LIN {X 0,Y 554.453,Z 809.786,A -85,B 0,C 180,E1 23627.307,E2 23627.307} C_VEL
LIN {X 0,Y 557.118,Z 789.157,A -85,B 0,C 180,E1 23626.499,E2 23626.499} C_VEL
LIN {X 0,Y 559.409,Z 768.857,A -85,B 0,C 180,E1 23625.833,E2 23625.833} C_VEL
LIN {X 0,Y 561.829,Z 743.404,A -85,B 0,C 180,E1 23625.168,E2 23625.168} C_VEL
LIN {X 0,Y 563.453,Z 718.234,A -85,B 0,C 180,E1 23624.694,E2 23624.694} C_VEL
LIN {X 0,Y 571.021,Z 495.759,A -85,B 0,C 180,E1 23621.491,E2 23621.491} C_VEL
LIN {X 0,Y 575.269,Z 370.947,A -85,B 0,C 180,E1 23619.667,E2 23619.667} C_VEL
LIN {X 0,Y 560.09,Z 346.765,A -85,B 0,C 180,E1 23617.356,E2 23617.356} C_VEL
LIN {X 0,Y 547.087,Z 327.659,A -85,B 0,C 180,E1 23615.214,E2 23615.214} C_VEL
LIN {X 0,Y 534.986,Z 310.945,A -85,B 0,C 180,E1 23613.044,E2 23613.044} C_VEL
LIN {X 0,Y 528.375,Z 302.282,A -85,B 0,C 180,E1 23611.773,E2 23611.773} C_VEL
LIN {X 0,Y 524.681,Z 297.482,A -85,B 0,C 180,E1 23611.031,E2 23611.031} C_VEL
LIN {X 0,Y 520.373,Z 291.905,A -85,B 0,C 180,E1 23610.132,E2 23610.132} C_VEL
LIN {X 0,Y 514.951,Z 285.155,A -85,B 0,C 180,E1 23608.914,E2 23608.914} C_VEL
LIN {X 0,Y 513.768,Z 282.099,A -85,B 0,C 180,E1 23608.162,E2 23608.162} C_VEL
LIN {X 0,Y 513.798,Z 281.966,A -85,B 0,C 180,E1 23604.857,E2 23604.857} C_VEL
LIN {X 0,Y 513.742,Z 281.98,A -85,B 0,C 180,E1 23601.583,E2 23601.583} C_VEL
LIN {X 0,Y 513.762,Z 281.984,A -85,B 0,C 180,E1 23598.143,E2 23598.143} C_VEL
LIN {X 0,Y 513.802,Z 281.979,A -85,B 0,C 180,E1 23594.719,E2 23594.719} C_VEL
LIN {X 0,Y 513.743,Z 281.974,A -85,B 0,C 180,E1 23591.337,E2 23591.337} C_VEL
LIN {X 0,Y 513.747,Z 281.962,A -85,B 0,C 180,E1 23587.83,E2 23587.83} C_VEL
LIN {X 0,Y 513.79,Z 281.955,A -85,B 0,C 180,E1 23584.577,E2 23584.577} C_VEL
LIN {X 0,Y 513.742,Z 281.977,A -85,B 0,C 180,E1 23581.227,E2 23581.227} C_VEL
LIN {X 0,Y 513.756,Z 281.987,A -85,B 0,C 180,E1 23577.769,E2 23577.769} C_VEL
LIN {X 0,Y 513.801,Z 281.966,A -85,B 0,C 180,E1 23574.304,E2 23574.304} C_VEL
LIN {X 0,Y 513.739,Z 281.958,A -85,B 0,C 180,E1 23571.042,E2 23571.042} C_VEL
LIN {X 0,Y 513.749,Z 281.959,A -85,B 0,C 180,E1 23567.524,E2 23567.524} C_VEL
LIN {X 0,Y 513.799,Z 281.966,A -85,B 0,C 180,E1 23564.19,E2 23564.19} C_VEL
LIN {X 0,Y 513.746,Z 281.987,A -85,B 0,C 180,E1 23560.797,E2 23560.797} C_VEL
LIN {X 0,Y 513.747,Z 281.987,A -85,B 0,C 180,E1 23557.213,E2 23557.213} C_VEL
LIN {X 0,Y 513.787,Z 281.879,A -85,B 0,C 180,E1 23553.907,E2 23553.907} C_VEL
LIN {X 0,Y 513.743,Z 281.964,A -85,B 0,C 180,E1 23550.629,E2 23550.629} C_VEL
LIN {X 0,Y 513.776,Z 282.125,A -85,B 0,C 180,E1 23548.389,E2 23548.389} C_VEL
LIN {X 0,Y 514.13,Z 283.467,A -85,B 0,C 180,E1 23548.085,E2 23548.085} C_VEL
LIN {X 0,Y 516.016,Z 286.518,A -85,B 0,C 180,E1 23547.636,E2 23547.636} C_VEL
LIN {X 0,Y 518.738,Z 288.732,A -85,B 0,C 180,E1 23547.073,E2 23547.073} C_VEL
LIN {X 0,Y 521.096,Z 292.417,A -85,B 0,C 180,E1 23546.552,E2 23546.552} C_VEL
LIN {X 0,Y 523.689,Z 294.869,A -85,B 0,C 180,E1 23546.033,E2 23546.033} C_VEL
LIN {X 0,Y 526.696,Z 298.998,A -85,B 0,C 180,E1 23545.415,E2 23545.415} C_VEL
LIN {X 0,Y 528.665,Z 301.077,A -85,B 0,C 180,E1 23545.035,E2 23545.035} C_VEL
LIN {X 0,Y 532.356,Z 305.607,A -85,B 0,C 180,E1 23544.324,E2 23544.324} C_VEL
LIN {X 0,Y 537,Z 311.379,A -85,B 0,C 180,E1 23543.461,E2 23543.461} C_VEL
LIN {X 0,Y 547.46,Z 325.856,A -85,B 0,C 180,E1 23541.594,E2 23541.594} C_VEL
LIN {X 0,Y 559.237,Z 342.837,A -85,B 0,C 180,E1 23539.649,E2 23539.649} C_VEL
LIN {X 0,Y 572.432,Z 363.406,A -85,B 0,C 180,E1 23537.625,E2 23537.625} C_VEL
LIN {X 0,Y 575.353,Z 368.355,A -85,B 0,C 180,E1 23537.193,E2 23537.193} C_VEL
LIN {X 0,Y 568.04,Z 579.703,A -85,B 0,C 180,E1 23534.136,E2 23534.136} C_VEL
LIN {X 0,Y 563.485,Z 712.252,A -85,B 0,C 180,E1 23532.221,E2 23532.221} C_VEL
LIN {X 0,Y 561.614,Z 739.268,A -85,B 0,C 180,E1 23531.688,E2 23531.688} C_VEL
LIN {X 0,Y 559.393,Z 762.648,A -85,B 0,C 180,E1 23531.056,E2 23531.056} C_VEL
LIN {X 0,Y 557.101,Z 783.032,A -85,B 0,C 180,E1 23530.373,E2 23530.373} C_VEL
LIN {X 0,Y 555.447,Z 790.439,A -85,B 0,C 180,E1 23530.171,E2 23530.171} C_VEL
LIN {X 0,Y 548.34,Z 809.024,A -85,B 0,C 180,E1 23529.808,E2 23529.808} C_VEL
LIN {X 0,Y 546.528,Z 815.961,A -85,B 0,C 180,E1 23529.545,E2 23529.545} C_VEL
LIN {X 0,Y 542.785,Z 839.215,A -85,B 0,C 180,E1 23528.327,E2 23528.327} C_VEL
LIN {X 0,Y 538.67,Z 861.769,A -85,B 0,C 180,E1 23526.911,E2 23526.911} C_VEL
LIN {X 0,Y 535.119,Z 880.065,A -85,B 0,C 180,E1 23525.595,E2 23525.595} C_VEL
LIN {X 0,Y 530.917,Z 900.978,A -85,B 0,C 180,E1 23523.88,E2 23523.88} C_VEL
LIN {X 0,Y 526.661,Z 920.781,A -85,B 0,C 180,E1 23521.985,E2 23521.985} C_VEL
LIN {X 0,Y 523.184,Z 936.83,A -85,B 0,C 180,E1 23520.248,E2 23520.248} C_VEL
LIN {X 0,Y 519.3,Z 954.991,A -85,B 0,C 180,E1 23518.022,E2 23518.022} C_VEL
LIN {X 0,Y 515.864,Z 971.093,A -85,B 0,C 180,E1 23515.733,E2 23515.733} C_VEL
LIN {X 0,Y 513.206,Z 984.016,A -85,B 0,C 180,E1 23513.663,E2 23513.663} C_VEL
LIN {X 0,Y 510.445,Z 998.558,A -85,B 0,C 180,E1 23511.006,E2 23511.006} C_VEL
LIN {X 0,Y 508.335,Z 1010.476,A -85,B 0,C 180,E1 23508.462,E2 23508.462} C_VEL
LIN {X 0,Y 506.857,Z 1020.106,A -85,B 0,C 180,E1 23506.112,E2 23506.112} C_VEL
LIN {X 0,Y 505.518,Z 1030.455,A -85,B 0,C 180,E1 23503.148,E2 23503.148} C_VEL
LIN {X 0,Y 504.78,Z 1037.728,A -85,B 0,C 180,E1 23500.615,E2 23500.615} C_VEL
LIN {X 0,Y 504.322,Z 1043.483,A -85,B 0,C 180,E1 23498.207,E2 23498.207} C_VEL
LIN {X 0,Y 504.05,Z 1048.716,A -85,B 0,C 180,E1 23495.464,E2 23495.464} C_VEL
LIN {X 0,Y 503.926,Z 1052.486,A -85,B 0,C 180,E1 23492.616,E2 23492.616} C_VEL
LIN {X 0,Y 503.916,Z 1054.489,A -85,B 0,C 180,E1 23490.227,E2 23490.227} C_VEL
LIN {X 0,Y 503.906,Z 1055.407,A -85,B 0,C 180,E1 23487.953,E2 23487.953} C_VEL
LIN {X 0,Y 503.904,Z 1055.329,A -85,B 0,C 180,E1 23485.562,E2 23485.562} C_VEL
LIN {X 0,Y 503.914,Z 1053.882,A -85,B 0,C 180,E1 23482.704,E2 23482.704} C_VEL
LIN {X 0,Y 503.979,Z 1050.859,A -85,B 0,C 180,E1 23479.945,E2 23479.945} C_VEL
LIN {X 0,Y 504.123,Z 1047.055,A -85,B 0,C 180,E1 23477.514,E2 23477.514} C_VEL
LIN {X 0,Y 504.455,Z 1041.841,A -85,B 0,C 180,E1 23474.95,E2 23474.95} C_VEL
LIN {X 0,Y 505.157,Z 1033.874,A -85,B 0,C 180,E1 23471.895,E2 23471.895} C_VEL
LIN {X 0,Y 506.062,Z 1025.946,A -85,B 0,C 180,E1 23469.409,E2 23469.409} C_VEL
LIN {X 0,Y 507.375,Z 1016.657,A -85,B 0,C 180,E1 23466.91,E2 23466.91} C_VEL
LIN {X 0,Y 509.449,Z 1003.972,A -85,B 0,C 180,E1 23464.016,E2 23464.016} C_VEL
LIN {X 0,Y 511.536,Z 992.584,A -85,B 0,C 180,E1 23461.769,E2 23461.769} C_VEL
LIN {X 0,Y 514.287,Z 978.894,A -85,B 0,C 180,E1 23459.377,E2 23459.377} C_VEL
LIN {X 0,Y 517.779,Z 962.343,A -85,B 0,C 180,E1 23456.873,E2 23456.873} C_VEL
LIN {X 0,Y 520.999,Z 947.641,A -85,B 0,C 180,E1 23454.915,E2 23454.915} C_VEL
LIN {X 0,Y 524.8,Z 930.682,A -85,B 0,C 180,E1 23452.906,E2 23452.906} C_VEL
LIN {X 0,Y 529.269,Z 910.241,A -85,B 0,C 180,E1 23450.807,E2 23450.807} C_VEL
LIN {X 0,Y 533.009,Z 892.867,A -85,B 0,C 180,E1 23449.245,E2 23449.245} C_VEL
LIN {X 0,Y 537.423,Z 871.919,A -85,B 0,C 180,E1 23447.59,E2 23447.59} C_VEL
LIN {X 0,Y 541.641,Z 850.035,A -85,B 0,C 180,E1 23446.117,E2 23446.117} C_VEL
LIN {X 0,Y 545.084,Z 830.856,A -85,B 0,C 180,E1 23444.997,E2 23444.997} C_VEL
LIN {X 0,Y 548.736,Z 808.878,A -85,B 0,C 180,E1 23443.891,E2 23443.891} C_VEL
LIN {X 0,Y 552.207,Z 784.715,A -85,B 0,C 180,E1 23442.885,E2 23442.885} C_VEL
LIN {X 0,Y 554.847,Z 763.158,A -85,B 0,C 180,E1 23442.15,E2 23442.15} C_VEL
LIN {X 0,Y 557.173,Z 740.46,A -85,B 0,C 180,E1 23441.525,E2 23441.525} C_VEL
LIN {X 0,Y 559.277,Z 712.892,A -85,B 0,C 180,E1 23440.968,E2 23440.968} C_VEL
LIN {X 0,Y 563.361,Z 607.457,A -85,B 0,C 180,E1 23439.413,E2 23439.413} C_VEL
LIN {X 0,Y 571.302,Z 402.325,A -85,B 0,C 180,E1 23436.395,E2 23436.395} C_VEL
LIN {X 0,Y 572.427,Z 372.307,A -85,B 0,C 180,E1 23435.938,E2 23435.938} C_VEL
LIN {X 0,Y 562.587,Z 356.836,A -85,B 0,C 180,E1 23434.292,E2 23434.292} C_VEL
LIN {X 0,Y 552.342,Z 341.781,A -85,B 0,C 180,E1 23432.463,E2 23432.463} C_VEL
LIN {X 0,Y 541.602,Z 326.838,A -85,B 0,C 180,E1 23430.388,E2 23430.388} C_VEL
LIN {X 0,Y 534.491,Z 317.842,A -85,B 0,C 180,E1 23428.92,E2 23428.92} C_VEL
LIN {X 0,Y 530.838,Z 313.286,A -85,B 0,C 180,E1 23428.124,E2 23428.124} C_VEL
LIN {X 0,Y 527.164,Z 308.769,A -85,B 0,C 180,E1 23427.293,E2 23427.293} C_VEL
LIN {X 0,Y 522.625,Z 303.55,A -85,B 0,C 180,E1 23426.229,E2 23426.229} C_VEL
LIN {X 0,Y 521.397,Z 301.779,A -85,B 0,C 180,E1 23425.92,E2 23425.92} C_VEL
LIN {X 0,Y 518.037,Z 298.4,A -85,B 0,C 180,E1 23425.097,E2 23425.097} C_VEL
LIN {X 0,Y 516.427,Z 295.827,A -85,B 0,C 180,E1 23424.661,E2 23424.661} C_VEL
LIN {X 0,Y 513.235,Z 293.149,A -85,B 0,C 180,E1 23423.845,E2 23423.845} C_VEL
LIN {X 0,Y 511.085,Z 289.592,A -85,B 0,C 180,E1 23423.217,E2 23423.217} C_VEL
LIN {X 0,Y 507.836,Z 287.317,A -85,B 0,C 180,E1 23422.334,E2 23422.334} C_VEL
LIN {X 0,Y 506.002,Z 283.836,A -85,B 0,C 180,E1 23421.686,E2 23421.686} C_VEL
LIN {X 0,Y 505.81,Z 282.987,A -85,B 0,C 180,E1 23421.208,E2 23421.208} C_VEL
LIN {X 0,Y 505.854,Z 282.932,A -85,B 0,C 180,E1 23417.841,E2 23417.841} C_VEL
LIN {X 0,Y 505.802,Z 282.897,A -85,B 0,C 180,E1 23414.54,E2 23414.54} C_VEL
LIN {X 0,Y 505.804,Z 282.954,A -85,B 0,C 180,E1 23411.055,E2 23411.055} C_VEL
LIN {X 0,Y 505.863,Z 282.882,A -85,B 0,C 180,E1 23407.724,E2 23407.724} C_VEL
LIN {X 0,Y 505.812,Z 282.949,A -85,B 0,C 180,E1 23404.308,E2 23404.308} C_VEL
LIN {X 0,Y 505.793,Z 282.891,A -85,B 0,C 180,E1 23400.793,E2 23400.793} C_VEL
LIN {X 0,Y 505.852,Z 282.939,A -85,B 0,C 180,E1 23397.508,E2 23397.508} C_VEL
LIN {X 0,Y 505.802,Z 282.898,A -85,B 0,C 180,E1 23394.214,E2 23394.214} C_VEL
LIN {X 0,Y 505.799,Z 282.933,A -85,B 0,C 180,E1 23390.671,E2 23390.671} C_VEL
LIN {X 0,Y 505.849,Z 282.89,A -85,B 0,C 180,E1 23387.326,E2 23387.326} C_VEL
LIN {X 0,Y 505.807,Z 282.926,A -85,B 0,C 180,E1 23384.051,E2 23384.051} C_VEL
LIN {X 0,Y 505.8,Z 282.897,A -85,B 0,C 180,E1 23380.553,E2 23380.553} C_VEL
LIN {X 0,Y 505.867,Z 282.942,A -85,B 0,C 180,E1 23377.206,E2 23377.206} C_VEL
LIN {X 0,Y 505.888,Z 283.351,A -85,B 0,C 180,E1 23375.667,E2 23375.667} C_VEL
LIN {X 0,Y 506.575,Z 285.399,A -85,B 0,C 180,E1 23375.17,E2 23375.17} C_VEL
LIN {X 0,Y 508.745,Z 288.207,A -85,B 0,C 180,E1 23374.505,E2 23374.505} C_VEL
LIN {X 0,Y 510.733,Z 289.915,A -85,B 0,C 180,E1 23373.958,E2 23373.958} C_VEL
LIN {X 0,Y 514.994,Z 294.989,A -85,B 0,C 180,E1 23372.791,E2 23372.791} C_VEL
LIN {X 0,Y 520.334,Z 301.55,A -85,B 0,C 180,E1 23371.413,E2 23371.413} C_VEL
LIN {X 0,Y 524.051,Z 305.988,A -85,B 0,C 180,E1 23370.51,E2 23370.51} C_VEL
LIN {X 0,Y 533.967,Z 318.851,A -85,B 0,C 180,E1 23368.251,E2 23368.251} C_VEL
LIN {X 0,Y 541.359,Z 328.901,A -85,B 0,C 180,E1 23366.7,E2 23366.7} C_VEL
LIN {X 0,Y 550.777,Z 341.951,A -85,B 0,C 180,E1 23364.866,E2 23364.866} C_VEL
LIN {X 0,Y 563.419,Z 360.814,A -85,B 0,C 180,E1 23362.599,E2 23362.599} C_VEL
LIN {X 0,Y 572.579,Z 375.694,A -85,B 0,C 180,E1 23361.069,E2 23361.069} C_VEL
LIN {X 0,Y 563.489,Z 607.493,A -85,B 0,C 180,E1 23357.666,E2 23357.666} C_VEL
LIN {X 0,Y 559.152,Z 720.201,A -85,B 0,C 180,E1 23356.004,E2 23356.004} C_VEL
LIN {X 0,Y 557.029,Z 747.91,A -85,B 0,C 180,E1 23355.449,E2 23355.449} C_VEL
LIN {X 0,Y 554.683,Z 770.486,A -85,B 0,C 180,E1 23354.834,E2 23354.834} C_VEL
LIN {X 0,Y 552.215,Z 790.549,A -85,B 0,C 180,E1 23354.16,E2 23354.16} C_VEL
LIN {X 0,Y 548.962,Z 813.722,A -85,B 0,C 180,E1 23353.224,E2 23353.224} C_VEL
LIN {X 0,Y 545.173,Z 836.653,A -85,B 0,C 180,E1 23352.094,E2 23352.094} C_VEL
LIN {X 0,Y 541.804,Z 855.478,A -85,B 0,C 180,E1 23351.017,E2 23351.017} C_VEL
LIN {X 0,Y 538.226,Z 874.224,A -85,B 0,C 180,E1 23349.791,E2 23349.791} C_VEL
LIN {X 0,Y 533.578,Z 897.113,A -85,B 0,C 180,E1 23348.062,E2 23348.062} C_VEL
LIN {X 0,Y 529.676,Z 915.321,A -85,B 0,C 180,E1 23346.469,E2 23346.469} C_VEL
LIN {X 0,Y 525.936,Z 932.493,A -85,B 0,C 180,E1 23344.774,E2 23344.774} C_VEL
LIN {X 0,Y 521.701,Z 951.969,A -85,B 0,C 180,E1 23342.586,E2 23342.586} C_VEL
LIN {X 0,Y 518.183,Z 968.123,A -85,B 0,C 180,E1 23340.496,E2 23340.496} C_VEL
LIN {X 0,Y 515.146,Z 982.591,A -85,B 0,C 180,E1 23338.394,E2 23338.394} C_VEL
LIN {X 0,Y 511.931,Z 998.836,A -85,B 0,C 180,E1 23335.696,E2 23335.696} C_VEL
LIN {X 0,Y 509.659,Z 1011.141,A -85,B 0,C 180,E1 23333.341,E2 23333.341} C_VEL
LIN {X 0,Y 507.902,Z 1021.942,A -85,B 0,C 180,E1 23330.996,E2 23330.996} C_VEL
LIN {X 0,Y 506.189,Z 1033.931,A -85,B 0,C 180,E1 23327.948,E2 23327.948} C_VEL
LIN {X 0,Y 505.253,Z 1042.032,A -85,B 0,C 180,E1 23325.495,E2 23325.495} C_VEL
LIN {X 0,Y 504.615,Z 1048.867,A -85,B 0,C 180,E1 23323.055,E2 23323.055} C_VEL
LIN {X 0,Y 504.158,Z 1055.624,A -85,B 0,C 180,E1 23320.051,E2 23320.051} C_VEL
LIN {X 0,Y 504,Z 1059.867,A -85,B 0,C 180,E1 23317.524,E2 23317.524} C_VEL
LIN {X 0,Y 503.923,Z 1062.669,A -85,B 0,C 180,E1 23315.237,E2 23315.237} C_VEL
LIN {X 0,Y 503.915,Z 1064.536,A -85,B 0,C 180,E1 23312.843,E2 23312.843} C_VEL
LIN {X 0,Y 503.913,Z 1065.403,A -85,B 0,C 180,E1 23310,E2 23310} C_VEL
LIN {X 0,Y 503.914,Z 1064.536,A -85,B 0,C 180,E1 23307.157,E2 23307.157} C_VEL
LIN {X 0,Y 503.923,Z 1062.669,A -85,B 0,C 180,E1 23304.763,E2 23304.763} C_VEL
LIN {X 0,Y 504.005,Z 1059.707,A -85,B 0,C 180,E1 23302.362,E2 23302.362} C_VEL
LIN {X 0,Y 504.219,Z 1054.753,A -85,B 0,C 180,E1 23299.488,E2 23299.488} C_VEL
LIN {X 0,Y 504.663,Z 1048.26,A -85,B 0,C 180,E1 23296.713,E2 23296.713} C_VEL
LIN {X 0,Y 505.289,Z 1041.681,A -85,B 0,C 180,E1 23294.388,E2 23294.388} C_VEL
LIN {X 0,Y 506.319,Z 1033.012,A -85,B 0,C 180,E1 23291.786,E2 23291.786} C_VEL
LIN {X 0,Y 507.978,Z 1021.444,A -85,B 0,C 180,E1 23288.887,E2 23288.887} C_VEL
LIN {X 0,Y 509.666,Z 1011.134,A -85,B 0,C 180,E1 23286.653,E2 23286.653} C_VEL
LIN {X 0,Y 511.933,Z 998.852,A -85,B 0,C 180,E1 23284.304,E2 23284.304} C_VEL
LIN {X 0,Y 515.136,Z 982.53,A -85,B 0,C 180,E1 23281.605,E2 23281.605} C_VEL
LIN {X 0,Y 517.974,Z 968.796,A -85,B 0,C 180,E1 23279.618,E2 23279.618} C_VEL
LIN {X 0,Y 521.233,Z 953.482,A -85,B 0,C 180,E1 23277.642,E2 23277.642} C_VEL
LIN {X 0,Y 525.45,Z 933.627,A -85,B 0,C 180,E1 23275.402,E2 23275.402} C_VEL
LIN {X 0,Y 529.03,Z 916.65,A -85,B 0,C 180,E1 23273.731,E2 23273.731} C_VEL
LIN {X 0,Y 532.787,Z 898.489,A -85,B 0,C 180,E1 23272.144,E2 23272.144} C_VEL
LIN {X 0,Y 537.401,Z 875.144,A -85,B 0,C 180,E1 23270.38,E2 23270.38} C_VEL
LIN {X 0,Y 540.935,Z 855.93,A -85,B 0,C 180,E1 23269.13,E2 23269.13} C_VEL
LIN {X 0,Y 544.258,Z 836.615,A -85,B 0,C 180,E1 23268.032,E2 23268.032} C_VEL
LIN {X 0,Y 548.122,Z 811.924,A -85,B 0,C 180,E1 23266.837,E2 23266.837} C_VEL
LIN {X 0,Y 551.03,Z 790.28,A -85,B 0,C 180,E1 23265.974,E2 23265.974} C_VEL
LIN {X 0,Y 553.399,Z 770.117,A -85,B 0,C 180,E1 23265.303,E2 23265.303} C_VEL
LIN {X 0,Y 555.717,Z 746.778,A -85,B 0,C 180,E1 23264.675,E2 23264.675} C_VEL
LIN {X 0,Y 557.645,Z 719.813,A -85,B 0,C 180,E1 23264.145,E2 23264.145} C_VEL
LIN {X 0,Y 562.993,Z 569.232,A -85,B 0,C 180,E1 23261.957,E2 23261.957} C_VEL
LIN {X 0,Y 569.951,Z 374.77,A -85,B 0,C 180,E1 23259.119,E2 23259.119} C_VEL
LIN {X 0,Y 555.897,Z 352.262,A -85,B 0,C 180,E1 23256.925,E2 23256.925} C_VEL
LIN {X 0,Y 543.365,Z 333.687,A -85,B 0,C 180,E1 23254.814,E2 23254.814} C_VEL
LIN {X 0,Y 531.41,Z 317,A -85,B 0,C 180,E1 23252.621,E2 23252.621} C_VEL
LIN {X 0,Y 524.88,Z 308.402,A -85,B 0,C 180,E1 23251.337,E2 23251.337} C_VEL
LIN {X 0,Y 521.584,Z 304.102,A -85,B 0,C 180,E1 23250.659,E2 23250.659} C_VEL
LIN {X 0,Y 517.442,Z 298.685,A -85,B 0,C 180,E1 23249.777,E2 23249.777} C_VEL
LIN {X 0,Y 509.213,Z 288.567,A -85,B 0,C 180,E1 23247.925,E2 23247.925} C_VEL
LIN {X 0,Y 506.669,Z 285.635,A -85,B 0,C 180,E1 23247.312,E2 23247.312} C_VEL
LIN {X 0,Y 505.899,Z 283.213,A -85,B 0,C 180,E1 23246.784,E2 23246.784} C_VEL
LIN {X 0,Y 505.807,Z 282.953,A -85,B 0,C 180,E1 23243.474,E2 23243.474} C_VEL
LIN {X 0,Y 505.805,Z 282.952,A -85,B 0,C 180,E1 23239.878,E2 23239.878} C_VEL
LIN {X 0,Y 505.857,Z 282.943,A -85,B 0,C 180,E1 23236.533,E2 23236.533} C_VEL
LIN {X 0,Y 505.808,Z 282.954,A -85,B 0,C 180,E1 23233.257,E2 23233.257} C_VEL
LIN {X 0,Y 505.807,Z 282.967,A -85,B 0,C 180,E1 23229.788,E2 23229.788} C_VEL
LIN {X 0,Y 505.871,Z 282.967,A -85,B 0,C 180,E1 23226.469,E2 23226.469} C_VEL
LIN {X 0,Y 505.811,Z 282.958,A -85,B 0,C 180,E1 23223.06,E2 23223.06} C_VEL
LIN {X 0,Y 505.801,Z 282.948,A -85,B 0,C 180,E1 23219.547,E2 23219.547} C_VEL
LIN {X 0,Y 505.854,Z 282.945,A -85,B 0,C 180,E1 23216.26,E2 23216.26} C_VEL
LIN {X 0,Y 505.81,Z 282.971,A -85,B 0,C 180,E1 23212.909,E2 23212.909} C_VEL
LIN {X 0,Y 505.807,Z 282.976,A -85,B 0,C 180,E1 23209.406,E2 23209.406} C_VEL
LIN {X 0,Y 505.864,Z 282.949,A -85,B 0,C 180,E1 23206.046,E2 23206.046} C_VEL
LIN {X 0,Y 505.814,Z 282.947,A -85,B 0,C 180,E1 23202.633,E2 23202.633} C_VEL
LIN {X 0,Y 505.802,Z 282.948,A -85,B 0,C 180,E1 23199.155,E2 23199.155} C_VEL
LIN {X 0,Y 505.852,Z 282.915,A -85,B 0,C 180,E1 23195.847,E2 23195.847} C_VEL
LIN {X 0,Y 505.807,Z 282.879,A -85,B 0,C 180,E1 23192.446,E2 23192.446} C_VEL
LIN {X 0,Y 505.885,Z 283.108,A -85,B 0,C 180,E1 23189.964,E2 23189.964} C_VEL
LIN {X 0,Y 506.188,Z 284.461,A -85,B 0,C 180,E1 23189.644,E2 23189.644} C_VEL
LIN {X 0,Y 507.959,Z 287.469,A -85,B 0,C 180,E1 23189.183,E2 23189.183} C_VEL
LIN {X 0,Y 510.968,Z 289.763,A -85,B 0,C 180,E1 23188.517,E2 23188.517} C_VEL
LIN {X 0,Y 513.385,Z 293.549,A -85,B 0,C 180,E1 23187.945,E2 23187.945} C_VEL
LIN {X 0,Y 515.995,Z 295.955,A -85,B 0,C 180,E1 23187.388,E2 23187.388} C_VEL
LIN {X 0,Y 518.916,Z 299.969,A -85,B 0,C 180,E1 23186.747,E2 23186.747} C_VEL
LIN {X 0,Y 520.905,Z 301.993,A -85,B 0,C 180,E1 23186.34,E2 23186.34} C_VEL
LIN {X 0,Y 524.449,Z 306.505,A -85,B 0,C 180,E1 23185.61,E2 23185.61} C_VEL
LIN {X 0,Y 526.85,Z 309.592,A -85,B 0,C 180,E1 23185.129,E2 23185.129} C_VEL
LIN {X 0,Y 530.776,Z 314.451,A -85,B 0,C 180,E1 23184.368,E2 23184.368} C_VEL
LIN {X 0,Y 536.926,Z 322.269,A -85,B 0,C 180,E1 23183.222,E2 23183.222} C_VEL
LIN {X 0,Y 547.877,Z 337.772,A -85,B 0,C 180,E1 23181.279,E2 23181.279} C_VEL
LIN {X 0,Y 558.734,Z 354.056,A -85,B 0,C 180,E1 23179.487,E2 23179.487} C_VEL
LIN {X 0,Y 569.982,Z 371.818,A -85,B 0,C 180,E1 23177.754,E2 23177.754} C_VEL
LIN {X 0,Y 562.566,Z 578.071,A -85,B 0,C 180,E1 23174.749,E2 23174.749} C_VEL
LIN {X 0,Y 557.767,Z 712.284,A -85,B 0,C 180,E1 23172.796,E2 23172.796} C_VEL
LIN {X 0,Y 555.852,Z 739.196,A -85,B 0,C 180,E1 23172.263,E2 23172.263} C_VEL
LIN {X 0,Y 553.559,Z 762.585,A -85,B 0,C 180,E1 23171.628,E2 23171.628} C_VEL
LIN {X 0,Y 551.1,Z 783.671,A -85,B 0,C 180,E1 23170.918,E2 23170.918} C_VEL
LIN {X 0,Y 547.756,Z 808.18,A -85,B 0,C 180,E1 23169.914,E2 23169.914} C_VEL
LIN {X 0,Y 546.528,Z 815.961,A -85,B 0,C 180,E1 23169.545,E2 23169.545} C_VEL
LIN {X 0,Y 544.695,Z 823.17,A -85,B 0,C 180,E1 23169.267,E2 23169.267} C_VEL
LIN {X 0,Y 537.052,Z 841.058,A -85,B 0,C 180,E1 23168.715,E2 23168.715} C_VEL
LIN {X 0,Y 535.041,Z 847.674,A -85,B 0,C 180,E1 23168.378,E2 23168.378} C_VEL
LIN {X 0,Y 531.464,Z 866.376,A -85,B 0,C 180,E1 23167.151,E2 23167.151} C_VEL
LIN {X 0,Y 526.686,Z 889.643,A -85,B 0,C 180,E1 23165.382,E2 23165.382} C_VEL
LIN {X 0,Y 522.685,Z 908.053,A -85,B 0,C 180,E1 23163.756,E2 23163.756} C_VEL
LIN {X 0,Y 518.678,Z 926.111,A -85,B 0,C 180,E1 23161.949,E2 23161.949} C_VEL
LIN {X 0,Y 514.32,Z 945.439,A -85,B 0,C 180,E1 23159.719,E2 23159.719} C_VEL
LIN {X 0,Y 510.958,Z 960.33,A -85,B 0,C 180,E1 23157.758,E2 23157.758} C_VEL
LIN {X 0,Y 507.691,Z 975.222,A -85,B 0,C 180,E1 23155.551,E2 23155.551} C_VEL
LIN {X 0,Y 504.387,Z 990.91,A -85,B 0,C 180,E1 23152.864,E2 23152.864} C_VEL
LIN {X 0,Y 502.139,Z 1002.299,A -85,B 0,C 180,E1 23150.626,E2 23150.626} C_VEL
LIN {X 0,Y 500.194,Z 1013.298,A -85,B 0,C 180,E1 23148.17,E2 23148.17} C_VEL
LIN {X 0,Y 498.438,Z 1024.538,A -85,B 0,C 180,E1 23145.222,E2 23145.222} C_VEL
LIN {X 0,Y 497.418,Z 1032.418,A -85,B 0,C 180,E1 23142.775,E2 23142.775} C_VEL
LIN {X 0,Y 496.721,Z 1039.128,A -85,B 0,C 180,E1 23140.32,E2 23140.32} C_VEL
LIN {X 0,Y 496.214,Z 1045.826,A -85,B 0,C 180,E1 23137.293,E2 23137.293} C_VEL
LIN {X 0,Y 496.013,Z 1050.189,A -85,B 0,C 180,E1 23134.625,E2 23134.625} C_VEL
LIN {X 0,Y 495.927,Z 1052.949,A -85,B 0,C 180,E1 23132.311,E2 23132.311} C_VEL
LIN {X 0,Y 495.929,Z 1054.797,A -85,B 0,C 180,E1 23129.884,E2 23129.884} C_VEL
LIN {X 0,Y 495.901,Z 1055.675,A -85,B 0,C 180,E1 23126.995,E2 23126.995} C_VEL
LIN {X 0,Y 495.917,Z 1054.841,A -85,B 0,C 180,E1 23124.098,E2 23124.098} C_VEL
LIN {X 0,Y 495.93,Z 1053.004,A -85,B 0,C 180,E1 23121.653,E2 23121.653} C_VEL
LIN {X 0,Y 496.014,Z 1050.23,A -85,B 0,C 180,E1 23119.312,E2 23119.312} C_VEL
LIN {X 0,Y 496.235,Z 1045.596,A -85,B 0,C 180,E1 23116.483,E2 23116.483} C_VEL
LIN {X 0,Y 496.712,Z 1039.241,A -85,B 0,C 180,E1 23113.631,E2 23113.631} C_VEL
LIN {X 0,Y 497.392,Z 1032.72,A -85,B 0,C 180,E1 23111.234,E2 23111.234} C_VEL
LIN {X 0,Y 498.37,Z 1025.03,A -85,B 0,C 180,E1 23108.83,E2 23108.83} C_VEL
LIN {X 0,Y 500.072,Z 1014.111,A -85,B 0,C 180,E1 23105.927,E2 23105.927} C_VEL
LIN {X 0,Y 502.055,Z 1002.775,A -85,B 0,C 180,E1 23103.378,E2 23103.378} C_VEL
LIN {X 0,Y 504.376,Z 991.131,A -85,B 0,C 180,E1 23101.072,E2 23101.072} C_VEL
LIN {X 0,Y 507.661,Z 975.743,A -85,B 0,C 180,E1 23098.405,E2 23098.405} C_VEL
LIN {X 0,Y 510.902,Z 961.281,A -85,B 0,C 180,E1 23096.233,E2 23096.233} C_VEL
LIN {X 0,Y 514.268,Z 946.705,A -85,B 0,C 180,E1 23094.282,E2 23094.282} C_VEL
LIN {X 0,Y 518.564,Z 928.403,A -85,B 0,C 180,E1 23092.112,E2 23092.112} C_VEL
LIN {X 0,Y 522.916,Z 909.332,A -85,B 0,C 180,E1 23090.166,E2 23090.166} C_VEL
LIN {X 0,Y 526.848,Z 891.87,A -85,B 0,C 180,E1 23088.593,E2 23088.593} C_VEL
LIN {X 0,Y 531.631,Z 869.908,A -85,B 0,C 180,E1 23086.866,E2 23086.866} C_VEL
LIN {X 0,Y 535.777,Z 849.121,A -85,B 0,C 180,E1 23085.472,E2 23085.472} C_VEL
LIN {X 0,Y 539.291,Z 830.262,A -85,B 0,C 180,E1 23084.37,E2 23084.37} C_VEL
LIN {X 0,Y 543.27,Z 807.157,A -85,B 0,C 180,E1 23083.21,E2 23083.21} C_VEL
LIN {X 0,Y 546.688,Z 783.707,A -85,B 0,C 180,E1 23082.245,E2 23082.245} C_VEL
LIN {X 0,Y 549.326,Z 762.831,A -85,B 0,C 180,E1 23081.534,E2 23081.534} C_VEL
LIN {X 0,Y 551.752,Z 739.902,A -85,B 0,C 180,E1 23080.904,E2 23080.904} C_VEL
LIN {X 0,Y 553.865,Z 712.736,A -85,B 0,C 180,E1 23080.357,E2 23080.357} C_VEL
LIN {X 0,Y 558.681,Z 592.582,A -85,B 0,C 180,E1 23078.574,E2 23078.574} C_VEL
LIN {X 0,Y 566.909,Z 389.826,A -85,B 0,C 180,E1 23075.57,E2 23075.57} C_VEL
LIN {X 0,Y 567.347,Z 376.066,A -85,B 0,C 180,E1 23075.346,E2 23075.346} C_VEL
LIN {X 0,Y 554.416,Z 355.965,A -85,B 0,C 180,E1 23073.094,E2 23073.094} C_VEL
LIN {X 0,Y 542.825,Z 339.313,A -85,B 0,C 180,E1 23070.895,E2 23070.895} C_VEL
LIN {X 0,Y 532.629,Z 325.707,A -85,B 0,C 180,E1 23068.785,E2 23068.785} C_VEL
LIN {X 0,Y 528,Z 320.103,A -85,B 0,C 180,E1 23067.766,E2 23067.766} C_VEL
LIN {X 0,Y 523.53,Z 314.602,A -85,B 0,C 180,E1 23066.73,E2 23066.73} C_VEL
LIN {X 0,Y 519.813,Z 310.104,A -85,B 0,C 180,E1 23065.829,E2 23065.829} C_VEL
LIN {X 0,Y 517.971,Z 308.142,A -85,B 0,C 180,E1 23065.376,E2 23065.376} C_VEL
LIN {X 0,Y 514.732,Z 304.072,A -85,B 0,C 180,E1 23064.533,E2 23064.533} C_VEL
LIN {X 0,Y 513.66,Z 302.878,A -85,B 0,C 180,E1 23064.251,E2 23064.251} C_VEL
LIN {X 0,Y 510.477,Z 299.652,A -85,B 0,C 180,E1 23063.399,E2 23063.399} C_VEL
LIN {X 0,Y 508.787,Z 297,A -85,B 0,C 180,E1 23062.9,E2 23062.9} C_VEL
LIN {X 0,Y 505.614,Z 294.456,A -85,B 0,C 180,E1 23062.009,E2 23062.009} C_VEL
LIN {X 0,Y 503.293,Z 290.628,A -85,B 0,C 180,E1 23061.258,E2 23061.258} C_VEL
LIN {X 0,Y 499.95,Z 288.31,A -85,B 0,C 180,E1 23060.243,E2 23060.243} C_VEL
LIN {X 0,Y 498.036,Z 284.769,A -85,B 0,C 180,E1 23059.468,E2 23059.468} C_VEL
LIN {X 0,Y 497.865,Z 283.951,A -85,B 0,C 180,E1 23058.865,E2 23058.865} C_VEL
LIN {X 0,Y 497.873,Z 283.902,A -85,B 0,C 180,E1 23055.373,E2 23055.373} C_VEL
LIN {X 0,Y 497.913,Z 283.897,A -85,B 0,C 180,E1 23051.937,E2 23051.937} C_VEL
LIN {X 0,Y 497.86,Z 283.894,A -85,B 0,C 180,E1 23048.547,E2 23048.547} C_VEL
LIN {X 0,Y 497.861,Z 283.908,A -85,B 0,C 180,E1 23044.954,E2 23044.954} C_VEL
LIN {X 0,Y 497.914,Z 283.888,A -85,B 0,C 180,E1 23041.611,E2 23041.611} C_VEL
LIN {X 0,Y 497.866,Z 283.899,A -85,B 0,C 180,E1 23038.274,E2 23038.274} C_VEL
LIN {X 0,Y 497.862,Z 283.902,A -85,B 0,C 180,E1 23034.815,E2 23034.815} C_VEL
LIN {X 0,Y 497.915,Z 283.883,A -85,B 0,C 180,E1 23031.454,E2 23031.454} C_VEL
LIN {X 0,Y 497.864,Z 283.907,A -85,B 0,C 180,E1 23028.179,E2 23028.179} C_VEL
LIN {X 0,Y 497.859,Z 283.894,A -85,B 0,C 180,E1 23024.583,E2 23024.583} C_VEL
LIN {X 0,Y 497.913,Z 283.893,A -85,B 0,C 180,E1 23021.258,E2 23021.258} C_VEL
LIN {X 0,Y 497.871,Z 283.985,A -85,B 0,C 180,E1 23018.065,E2 23018.065} C_VEL
LIN {X 0,Y 498.088,Z 284.909,A -85,B 0,C 180,E1 23017.578,E2 23017.578} C_VEL
LIN {X 0,Y 499.92,Z 288.355,A -85,B 0,C 180,E1 23016.857,E2 23016.857} C_VEL
LIN {X 0,Y 503.598,Z 291.248,A -85,B 0,C 180,E1 23015.732,E2 23015.732} C_VEL
LIN {X 0,Y 506.149,Z 295.077,A -85,B 0,C 180,E1 23014.929,E2 23014.929} C_VEL
LIN {X 0,Y 508.844,Z 297.566,A -85,B 0,C 180,E1 23014.167,E2 23014.167} C_VEL
LIN {X 0,Y 517.763,Z 308.441,A -85,B 0,C 180,E1 23011.762,E2 23011.762} C_VEL
LIN {X 0,Y 522.961,Z 315.065,A -85,B 0,C 180,E1 23010.474,E2 23010.474} C_VEL
LIN {X 0,Y 530.46,Z 324.682,A -85,B 0,C 180,E1 23008.746,E2 23008.746} C_VEL
LIN {X 0,Y 538.88,Z 336.291,A -85,B 0,C 180,E1 23006.94,E2 23006.94} C_VEL
LIN {X 0,Y 547.737,Z 348.715,A -85,B 0,C 180,E1 23005.185,E2 23005.185} C_VEL
LIN {X 0,Y 560.312,Z 367.704,A -85,B 0,C 180,E1 23002.887,E2 23002.887} C_VEL
LIN {X 0,Y 567.522,Z 379.675,A -85,B 0,C 180,E1 23001.65,E2 23001.65} C_VEL
LIN {X 0,Y 558.027,Z 612.752,A -85,B 0,C 180,E1 22998.208,E2 22998.208} C_VEL
LIN {X 0,Y 553.713,Z 720.242,A -85,B 0,C 180,E1 22996.612,E2 22996.612} C_VEL
LIN {X 0,Y 551.502,Z 748.093,A -85,B 0,C 180,E1 22996.049,E2 22996.049} C_VEL
LIN {X 0,Y 549.117,Z 770.299,A -85,B 0,C 180,E1 22995.442,E2 22995.442} C_VEL
LIN {X 0,Y 546.582,Z 790.192,A -85,B 0,C 180,E1 22994.773,E2 22994.773} C_VEL
LIN {X 0,Y 543.114,Z 814.028,A -85,B 0,C 180,E1 22993.806,E2 22993.806} C_VEL
LIN {X 0,Y 539.188,Z 836.876,A -85,B 0,C 180,E1 22992.671,E2 22992.671} C_VEL
LIN {X 0,Y 535.698,Z 855.615,A -85,B 0,C 180,E1 22991.591,E2 22991.591} C_VEL
LIN {X 0,Y 531.812,Z 875.187,A -85,B 0,C 180,E1 22990.299,E2 22990.299} C_VEL
LIN {X 0,Y 526.83,Z 898.55,A -85,B 0,C 180,E1 22988.5,E2 22988.5} C_VEL
LIN {X 0,Y 522.829,Z 916.457,A -85,B 0,C 180,E1 22986.906,E2 22986.906} C_VEL
LIN {X 0,Y 518.79,Z 934.215,A -85,B 0,C 180,E1 22985.121,E2 22985.121} C_VEL
LIN {X 0,Y 514.173,Z 954.309,A -85,B 0,C 180,E1 22982.792,E2 22982.792} C_VEL
LIN {X 0,Y 510.838,Z 968.976,A -85,B 0,C 180,E1 22980.852,E2 22980.852} C_VEL
LIN {X 0,Y 507.512,Z 984.119,A -85,B 0,C 180,E1 22978.604,E2 22978.604} C_VEL
LIN {X 0,Y 504.302,Z 999.426,A -85,B 0,C 180,E1 22975.988,E2 22975.988} C_VEL
LIN {X 0,Y 502.045,Z 1011.037,A -85,B 0,C 180,E1 22973.723,E2 22973.723} C_VEL
LIN {X 0,Y 500.085,Z 1022.376,A -85,B 0,C 180,E1 22971.217,E2 22971.217} C_VEL
LIN {X 0,Y 498.35,Z 1033.848,A -85,B 0,C 180,E1 22968.24,E2 22968.24} C_VEL
LIN {X 0,Y 497.343,Z 1041.95,A -85,B 0,C 180,E1 22965.748,E2 22965.748} C_VEL
LIN {X 0,Y 496.667,Z 1048.786,A -85,B 0,C 180,E1 22963.268,E2 22963.268} C_VEL
LIN {X 0,Y 496.179,Z 1055.544,A -85,B 0,C 180,E1 22960.215,E2 22960.215} C_VEL
LIN {X 0,Y 496.006,Z 1059.788,A -85,B 0,C 180,E1 22957.646,E2 22957.646} C_VEL
LIN {X 0,Y 495.923,Z 1062.591,A -85,B 0,C 180,E1 22955.322,E2 22955.322} C_VEL
LIN {X 0,Y 495.914,Z 1064.458,A -85,B 0,C 180,E1 22952.889,E2 22952.889} C_VEL
LIN {X 0,Y 495.914,Z 1065.325,A -85,B 0,C 180,E1 22950,E2 22950} C_VEL
LIN {X 0,Y 495.914,Z 1064.458,A -85,B 0,C 180,E1 22947.111,E2 22947.111} C_VEL
LIN {X 0,Y 495.923,Z 1062.591,A -85,B 0,C 180,E1 22944.678,E2 22944.678} C_VEL
LIN {X 0,Y 496.006,Z 1059.79,A -85,B 0,C 180,E1 22942.354,E2 22942.354} C_VEL
LIN {X 0,Y 496.229,Z 1054.92,A -85,B 0,C 180,E1 22939.434,E2 22939.434} C_VEL
LIN {X 0,Y 496.692,Z 1048.486,A -85,B 0,C 180,E1 22936.614,E2 22936.614} C_VEL
LIN {X 0,Y 497.38,Z 1041.601,A -85,B 0,C 180,E1 22934.133,E2 22934.133} C_VEL
LIN {X 0,Y 498.468,Z 1033.045,A -85,B 0,C 180,E1 22931.522,E2 22931.522} C_VEL
LIN {X 0,Y 500.245,Z 1021.363,A -85,B 0,C 180,E1 22928.545,E2 22928.545} C_VEL
LIN {X 0,Y 502.046,Z 1011.049,A -85,B 0,C 180,E1 22926.278,E2 22926.278} C_VEL
LIN {X 0,Y 504.428,Z 998.73,A -85,B 0,C 180,E1 22923.89,E2 22923.89} C_VEL
LIN {X 0,Y 507.812,Z 982.385,A -85,B 0,C 180,E1 22921.157,E2 22921.157} C_VEL
LIN {X 0,Y 510.784,Z 968.629,A -85,B 0,C 180,E1 22919.144,E2 22919.144} C_VEL
LIN {X 0,Y 514.295,Z 952.828,A -85,B 0,C 180,E1 22917.085,E2 22917.085} C_VEL
LIN {X 0,Y 518.768,Z 932.721,A -85,B 0,C 180,E1 22914.809,E2 22914.809} C_VEL
LIN {X 0,Y 522.536,Z 915.604,A -85,B 0,C 180,E1 22913.117,E2 22913.117} C_VEL
LIN {X 0,Y 526.876,Z 895.527,A -85,B 0,C 180,E1 22911.365,E2 22911.365} C_VEL
LIN {X 0,Y 531.299,Z 873.578,A -85,B 0,C 180,E1 22909.725,E2 22909.725} C_VEL
LIN {X 0,Y 534.901,Z 854.676,A -85,B 0,C 180,E1 22908.497,E2 22908.497} C_VEL
LIN {X 0,Y 538.549,Z 834.205,A -85,B 0,C 180,E1 22907.338,E2 22907.338} C_VEL
LIN {X 0,Y 542.539,Z 808.858,A -85,B 0,C 180,E1 22906.135,E2 22906.135} C_VEL
LIN {X 0,Y 545.391,Z 788.253,A -85,B 0,C 180,E1 22905.325,E2 22905.325} C_VEL
LIN {X 0,Y 547.791,Z 768.364,A -85,B 0,C 180,E1 22904.672,E2 22904.672} C_VEL
LIN {X 0,Y 550.352,Z 742.96,A -85,B 0,C 180,E1 22904.005,E2 22904.005} C_VEL
LIN {X 0,Y 552.067,Z 717.9,A -85,B 0,C 180,E1 22903.529,E2 22903.529} C_VEL
LIN {X 0,Y 560.361,Z 493,A -85,B 0,C 180,E1 22900.244,E2 22900.244} C_VEL
LIN {X 0,Y 564.599,Z 378.505,A -85,B 0,C 180,E1 22898.548,E2 22898.548} C_VEL
LIN {X 0,Y 551.797,Z 357.871,A -85,B 0,C 180,E1 22896.499,E2 22896.499} C_VEL
LIN {X 0,Y 539.928,Z 340.063,A -85,B 0,C 180,E1 22894.455,E2 22894.455} C_VEL
LIN {X 0,Y 527.024,Z 321.828,A -85,B 0,C 180,E1 22892.024,E2 22892.024} C_VEL
LIN {X 0,Y 518.51,Z 310.703,A -85,B 0,C 180,E1 22890.283,E2 22890.283} C_VEL
LIN {X 0,Y 514.418,Z 305.324,A -85,B 0,C 180,E1 22889.393,E2 22889.393} C_VEL
LIN {X 0,Y 506.728,Z 295.743,A -85,B 0,C 180,E1 22887.627,E2 22887.627} C_VEL
LIN {X 0,Y 503.861,Z 292.349,A -85,B 0,C 180,E1 22886.933,E2 22886.933} C_VEL
LIN {X 0,Y 502.33,Z 290.191,A -85,B 0,C 180,E1 22886.543,E2 22886.543} C_VEL
LIN {X 0,Y 499.364,Z 287.714,A -85,B 0,C 180,E1 22885.818,E2 22885.818} C_VEL
LIN {X 0,Y 497.99,Z 284.608,A -85,B 0,C 180,E1 22885.32,E2 22885.32} C_VEL
LIN {X 0,Y 497.923,Z 283.958,A -85,B 0,C 180,E1 22884.816,E2 22884.816} C_VEL
LIN {X 0,Y 497.871,Z 283.951,A -85,B 0,C 180,E1 22881.44,E2 22881.44} C_VEL
LIN {X 0,Y 497.868,Z 283.955,A -85,B 0,C 180,E1 22877.834,E2 22877.834} C_VEL
LIN {X 0,Y 497.916,Z 283.96,A -85,B 0,C 180,E1 22874.419,E2 22874.419} C_VEL
LIN {X 0,Y 497.885,Z 283.956,A -85,B 0,C 180,E1 22870.999,E2 22870.999} C_VEL
LIN {X 0,Y 497.862,Z 283.943,A -85,B 0,C 180,E1 22867.501,E2 22867.501} C_VEL
LIN {X 0,Y 497.899,Z 283.931,A -85,B 0,C 180,E1 22864.146,E2 22864.146} C_VEL
LIN {X 0,Y 497.896,Z 283.937,A -85,B 0,C 180,E1 22860.69,E2 22860.69} C_VEL
LIN {X 0,Y 497.864,Z 283.962,A -85,B 0,C 180,E1 22857.237,E2 22857.237} C_VEL
LIN {X 0,Y 497.884,Z 283.959,A -85,B 0,C 180,E1 22853.768,E2 22853.768} C_VEL
LIN {X 0,Y 497.907,Z 283.935,A -85,B 0,C 180,E1 22850.405,E2 22850.405} C_VEL
LIN {X 0,Y 497.862,Z 283.935,A -85,B 0,C 180,E1 22847.001,E2 22847.001} C_VEL
LIN {X 0,Y 497.878,Z 283.937,A -85,B 0,C 180,E1 22843.55,E2 22843.55} C_VEL
LIN {X 0,Y 497.916,Z 283.941,A -85,B 0,C 180,E1 22840.161,E2 22840.161} C_VEL
LIN {X 0,Y 497.865,Z 283.956,A -85,B 0,C 180,E1 22836.819,E2 22836.819} C_VEL
LIN {X 0,Y 497.862,Z 283.855,A -85,B 0,C 180,E1 22833.264,E2 22833.264} C_VEL
LIN {X 0,Y 497.935,Z 284.133,A -85,B 0,C 180,E1 22831.646,E2 22831.646} C_VEL
LIN {X 0,Y 498.264,Z 285.571,A -85,B 0,C 180,E1 22831.323,E2 22831.323} C_VEL
LIN {X 0,Y 500.038,Z 288.49,A -85,B 0,C 180,E1 22830.829,E2 22830.829} C_VEL
LIN {X 0,Y 503.17,Z 290.859,A -85,B 0,C 180,E1 22830.08,E2 22830.08} C_VEL
LIN {X 0,Y 505.404,Z 294.504,A -85,B 0,C 180,E1 22829.505,E2 22829.505} C_VEL
LIN {X 0,Y 508.441,Z 297.204,A -85,B 0,C 180,E1 22828.81,E2 22828.81} C_VEL
LIN {X 0,Y 511.447,Z 301.282,A -85,B 0,C 180,E1 22828.106,E2 22828.106} C_VEL
LIN {X 0,Y 513.391,Z 303.233,A -85,B 0,C 180,E1 22827.682,E2 22827.682} C_VEL
LIN {X 0,Y 516.799,Z 307.548,A -85,B 0,C 180,E1 22826.934,E2 22826.934} C_VEL
LIN {X 0,Y 518.539,Z 309.672,A -85,B 0,C 180,E1 22826.564,E2 22826.564} C_VEL
LIN {X 0,Y 523.739,Z 316.174,A -85,B 0,C 180,E1 22825.491,E2 22825.491} C_VEL
LIN {X 0,Y 528.597,Z 322.348,A -85,B 0,C 180,E1 22824.532,E2 22824.532} C_VEL
LIN {X 0,Y 533.957,Z 329.222,A -85,B 0,C 180,E1 22823.519,E2 22823.519} C_VEL
LIN {X 0,Y 546.265,Z 346.772,A -85,B 0,C 180,E1 22821.311,E2 22821.311} C_VEL
LIN {X 0,Y 558.78,Z 366.158,A -85,B 0,C 180,E1 22819.238,E2 22819.238} C_VEL
LIN {X 0,Y 564.67,Z 375.819,A -85,B 0,C 180,E1 22818.314,E2 22818.314} C_VEL
LIN {X 0,Y 556.86,Z 584.496,A -85,B 0,C 180,E1 22815.256,E2 22815.256} C_VEL
LIN {X 0,Y 552.093,Z 712.5,A -85,B 0,C 180,E1 22813.379,E2 22813.379} C_VEL
LIN {X 0,Y 550.079,Z 739.75,A -85,B 0,C 180,E1 22812.834,E2 22812.834} C_VEL
LIN {X 0,Y 547.745,Z 762.81,A -85,B 0,C 180,E1 22812.204,E2 22812.204} C_VEL
LIN {X 0,Y 545.304,Z 783.096,A -85,B 0,C 180,E1 22811.518,E2 22811.518} C_VEL
LIN {X 0,Y 542.036,Z 806.648,A -85,B 0,C 180,E1 22810.56,E2 22810.56} C_VEL
LIN {X 0,Y 538.318,Z 829.27,A -85,B 0,C 180,E1 22809.438,E2 22809.438} C_VEL
LIN {X 0,Y 535.041,Z 847.674,A -85,B 0,C 180,E1 22808.378,E2 22808.378} C_VEL
LIN {X 0,Y 533.004,Z 854.583,A -85,B 0,C 180,E1 22808.026,E2 22808.026} C_VEL
LIN {X 0,Y 524.485,Z 872.536,A -85,B 0,C 180,E1 22807.232,E2 22807.232} C_VEL
LIN {X 0,Y 522.713,Z 877.924,A -85,B 0,C 180,E1 22806.871,E2 22806.871} C_VEL
LIN {X 0,Y 518.72,Z 896.239,A -85,B 0,C 180,E1 22805.375,E2 22805.375} C_VEL
LIN {X 0,Y 513.841,Z 917.786,A -85,B 0,C 180,E1 22803.348,E2 22803.348} C_VEL
LIN {X 0,Y 509.863,Z 934.706,A -85,B 0,C 180,E1 22801.509,E2 22801.509} C_VEL
LIN {X 0,Y 506.288,Z 949.842,A -85,B 0,C 180,E1 22799.66,E2 22799.66} C_VEL
LIN {X 0,Y 502.238,Z 967.226,A -85,B 0,C 180,E1 22797.251,E2 22797.251} C_VEL
LIN {X 0,Y 498.875,Z 981.918,A -85,B 0,C 180,E1 22794.891,E2 22794.891} C_VEL
LIN {X 0,Y 496.193,Z 994.332,A -85,B 0,C 180,E1 22792.637,E2 22792.637} C_VEL
LIN {X 0,Y 493.481,Z 1008.029,A -85,B 0,C 180,E1 22789.778,E2 22789.778} C_VEL
LIN {X 0,Y 491.626,Z 1018.259,A -85,B 0,C 180,E1 22787.274,E2 22787.274} C_VEL
LIN {X 0,Y 490.271,Z 1026.946,A -85,B 0,C 180,E1 22784.825,E2 22784.825} C_VEL
LIN {X 0,Y 489.168,Z 1035.757,A -85,B 0,C 180,E1 22781.914,E2 22781.914} C_VEL
LIN {X 0,Y 488.499,Z 1042.603,A -85,B 0,C 180,E1 22779.068,E2 22779.068} C_VEL
LIN {X 0,Y 488.15,Z 1047.454,A -85,B 0,C 180,E1 22776.564,E2 22776.564} C_VEL
LIN {X 0,Y 487.984,Z 1051.281,A -85,B 0,C 180,E1 22773.995,E2 22773.995} C_VEL
LIN {X 0,Y 487.923,Z 1054.297,A -85,B 0,C 180,E1 22770.939,E2 22770.939} C_VEL
LIN {X 0,Y 487.9,Z 1055.492,A -85,B 0,C 180,E1 22768.356,E2 22768.356} C_VEL
LIN {X 0,Y 487.904,Z 1055.579,A -85,B 0,C 180,E1 22766.004,E2 22766.004} C_VEL
LIN {X 0,Y 487.914,Z 1054.687,A -85,B 0,C 180,E1 22763.646,E2 22763.646} C_VEL
LIN {X 0,Y 487.933,Z 1052.694,A -85,B 0,C 180,E1 22761.159,E2 22761.159} C_VEL
LIN {X 0,Y 488.075,Z 1048.899,A -85,B 0,C 180,E1 22758.178,E2 22758.178} C_VEL
LIN {X 0,Y 488.388,Z 1043.822,A -85,B 0,C 180,E1 22755.415,E2 22755.415} C_VEL
LIN {X 0,Y 488.897,Z 1038.275,A -85,B 0,C 180,E1 22752.995,E2 22752.995} C_VEL
LIN {X 0,Y 489.694,Z 1031.233,A -85,B 0,C 180,E1 22750.436,E2 22750.436} C_VEL
LIN {X 0,Y 491.258,Z 1020.587,A -85,B 0,C 180,E1 22747.25,E2 22747.25} C_VEL
LIN {X 0,Y 492.949,Z 1010.815,A -85,B 0,C 180,E1 22744.778,E2 22744.778} C_VEL
LIN {X 0,Y 495.253,Z 999.165,A -85,B 0,C 180,E1 22742.201,E2 22742.201} C_VEL
LIN {X 0,Y 498.483,Z 984.228,A -85,B 0,C 180,E1 22739.37,E2 22739.37} C_VEL
LIN {X 0,Y 501.368,Z 971.671,A -85,B 0,C 180,E1 22737.285,E2 22737.285} C_VEL
LIN {X 0,Y 504.967,Z 956.623,A -85,B 0,C 180,E1 22735.062,E2 22735.062} C_VEL
LIN {X 0,Y 509.511,Z 937.96,A -85,B 0,C 180,E1 22732.671,E2 22732.671} C_VEL
LIN {X 0,Y 513.404,Z 921.965,A -85,B 0,C 180,E1 22730.875,E2 22730.875} C_VEL
LIN {X 0,Y 517.544,Z 904.74,A -85,B 0,C 180,E1 22729.158,E2 22729.158} C_VEL
LIN {X 0,Y 522.692,Z 882.387,A -85,B 0,C 180,E1 22727.227,E2 22727.227} C_VEL
LIN {X 0,Y 526.751,Z 863.801,A -85,B 0,C 180,E1 22725.842,E2 22725.842} C_VEL
LIN {X 0,Y 530.7,Z 844.601,A -85,B 0,C 180,E1 22724.587,E2 22724.587} C_VEL
LIN {X 0,Y 535.256,Z 820.382,A -85,B 0,C 180,E1 22723.236,E2 22723.236} C_VEL
LIN {X 0,Y 538.826,Z 798.817,A -85,B 0,C 180,E1 22722.233,E2 22722.233} C_VEL
LIN {X 0,Y 541.829,Z 778.473,A -85,B 0,C 180,E1 22721.437,E2 22721.437} C_VEL
LIN {X 0,Y 544.915,Z 754.145,A -85,B 0,C 180,E1 22720.653,E2 22720.653} C_VEL
LIN {X 0,Y 547.297,Z 729.225,A -85,B 0,C 180,E1 22720.049,E2 22720.049} C_VEL
LIN {X 0,Y 548.806,Z 707.403,A -85,B 0,C 180,E1 22719.648,E2 22719.648} C_VEL
LIN {X 0,Y 558.563,Z 472.044,A -85,B 0,C 180,E1 22716.153,E2 22716.153} C_VEL
LIN {X 0,Y 562.391,Z 380.014,A -85,B 0,C 180,E1 22714.755,E2 22714.755} C_VEL
LIN {X 0,Y 549.355,Z 359.739,A -85,B 0,C 180,E1 22712.414,E2 22712.414} C_VEL
LIN {X 0,Y 538.086,Z 343.721,A -85,B 0,C 180,E1 22710.207,E2 22710.207} C_VEL
LIN {X 0,Y 529.87,Z 332.596,A -85,B 0,C 180,E1 22708.456,E2 22708.456} C_VEL
LIN {X 0,Y 525.077,Z 326.78,A -85,B 0,C 180,E1 22707.38,E2 22707.38} C_VEL
LIN {X 0,Y 520.77,Z 321.454,A -85,B 0,C 180,E1 22706.36,E2 22706.36} C_VEL
LIN {X 0,Y 516.207,Z 315.866,A -85,B 0,C 180,E1 22705.223,E2 22705.223} C_VEL
LIN {X 0,Y 512.579,Z 311.55,A -85,B 0,C 180,E1 22704.275,E2 22704.275} C_VEL
LIN {X 0,Y 511.328,Z 310.123,A -85,B 0,C 180,E1 22703.939,E2 22703.939} C_VEL
LIN {X 0,Y 507.933,Z 306.386,A -85,B 0,C 180,E1 22703.002,E2 22703.002} C_VEL
LIN {X 0,Y 506.51,Z 304.375,A -85,B 0,C 180,E1 22702.579,E2 22702.579} C_VEL
LIN {X 0,Y 503.238,Z 301.366,A -85,B 0,C 180,E1 22701.628,E2 22701.628} C_VEL
LIN {X 0,Y 501.453,Z 298.252,A -85,B 0,C 180,E1 22701.034,E2 22701.034} C_VEL
LIN {X 0,Y 497.994,Z 295.663,A -85,B 0,C 180,E1 22699.958,E2 22699.958} C_VEL
LIN {X 0,Y 495.564,Z 291.78,A -85,B 0,C 180,E1 22699.079,E2 22699.079} C_VEL
LIN {X 0,Y 491.924,Z 289.226,A -85,B 0,C 180,E1 22697.813,E2 22697.813} C_VEL
LIN {X 0,Y 490.254,Z 286.418,A -85,B 0,C 180,E1 22697.11,E2 22697.11} C_VEL
LIN {X 0,Y 489.954,Z 285.098,A -85,B 0,C 180,E1 22696.601,E2 22696.601} C_VEL
LIN {X 0,Y 489.918,Z 284.866,A -85,B 0,C 180,E1 22693.094,E2 22693.094} C_VEL
LIN {X 0,Y 489.968,Z 284.918,A -85,B 0,C 180,E1 22689.633,E2 22689.633} C_VEL
LIN {X 0,Y 489.927,Z 284.86,A -85,B 0,C 180,E1 22686.326,E2 22686.326} C_VEL
LIN {X 0,Y 489.923,Z 284.928,A -85,B 0,C 180,E1 22682.808,E2 22682.808} C_VEL
LIN {X 0,Y 489.96,Z 284.855,A -85,B 0,C 180,E1 22679.415,E2 22679.415} C_VEL
LIN {X 0,Y 489.956,Z 284.932,A -85,B 0,C 180,E1 22675.904,E2 22675.904} C_VEL
LIN {X 0,Y 489.913,Z 284.858,A -85,B 0,C 180,E1 22672.494,E2 22672.494} C_VEL
LIN {X 0,Y 489.944,Z 284.928,A -85,B 0,C 180,E1 22669.001,E2 22669.001} C_VEL
LIN {X 0,Y 489.981,Z 284.853,A -85,B 0,C 180,E1 22665.463,E2 22665.463} C_VEL
LIN {X 0,Y 489.933,Z 284.91,A -85,B 0,C 180,E1 22661.997,E2 22661.997} C_VEL
LIN {X 0,Y 489.947,Z 285.077,A -85,B 0,C 180,E1 22660.446,E2 22660.446} C_VEL
LIN {X 0,Y 490.236,Z 286.292,A -85,B 0,C 180,E1 22660.001,E2 22660.001} C_VEL
LIN {X 0,Y 492.064,Z 289.331,A -85,B 0,C 180,E1 22659.232,E2 22659.232} C_VEL
LIN {X 0,Y 495.867,Z 292.104,A -85,B 0,C 180,E1 22657.91,E2 22657.91} C_VEL
LIN {X 0,Y 498.142,Z 295.911,A -85,B 0,C 180,E1 22657.082,E2 22657.082} C_VEL
LIN {X 0,Y 501.595,Z 298.712,A -85,B 0,C 180,E1 22656.005,E2 22656.005} C_VEL
LIN {X 0,Y 504.302,Z 302.631,A -85,B 0,C 180,E1 22655.144,E2 22655.144} C_VEL
LIN {X 0,Y 506.873,Z 305.078,A -85,B 0,C 180,E1 22654.404,E2 22654.404} C_VEL
LIN {X 0,Y 515.308,Z 315.481,A -85,B 0,C 180,E1 22652.088,E2 22652.088} C_VEL
LIN {X 0,Y 520.747,Z 322.531,A -85,B 0,C 180,E1 22650.715,E2 22650.715} C_VEL
LIN {X 0,Y 528.068,Z 332.033,A -85,B 0,C 180,E1 22649,E2 22649} C_VEL
LIN {X 0,Y 538.61,Z 346.621,A -85,B 0,C 180,E1 22646.731,E2 22646.731} C_VEL
LIN {X 0,Y 549.654,Z 362.899,A -85,B 0,C 180,E1 22644.56,E2 22644.56} C_VEL
LIN {X 0,Y 560.385,Z 379.764,A -85,B 0,C 180,E1 22642.619,E2 22642.619} C_VEL
LIN {X 0,Y 562.517,Z 383.702,A -85,B 0,C 180,E1 22642.242,E2 22642.242} C_VEL
LIN {X 0,Y 552.7,Z 615.883,A -85,B 0,C 180,E1 22638.792,E2 22638.792} C_VEL
LIN {X 0,Y 548.345,Z 720.199,A -85,B 0,C 180,E1 22637.232,E2 22637.232} C_VEL
LIN {X 0,Y 546.052,Z 748.162,A -85,B 0,C 180,E1 22636.665,E2 22636.665} C_VEL
LIN {X 0,Y 543.614,Z 770.126,A -85,B 0,C 180,E1 22636.062,E2 22636.062} C_VEL
LIN {X 0,Y 541.094,Z 789.259,A -85,B 0,C 180,E1 22635.42,E2 22635.42} C_VEL
LIN {X 0,Y 537.703,Z 811.81,A -85,B 0,C 180,E1 22634.511,E2 22634.511} C_VEL
LIN {X 0,Y 533.449,Z 836.11,A -85,B 0,C 180,E1 22633.316,E2 22633.316} C_VEL
LIN {X 0,Y 529.764,Z 855.173,A -85,B 0,C 180,E1 22632.215,E2 22632.215} C_VEL
LIN {X 0,Y 525.768,Z 874.545,A -85,B 0,C 180,E1 22630.931,E2 22630.931} C_VEL
LIN {X 0,Y 520.748,Z 897.336,A -85,B 0,C 180,E1 22629.176,E2 22629.176} C_VEL
LIN {X 0,Y 516.413,Z 915.921,A -85,B 0,C 180,E1 22627.515,E2 22627.515} C_VEL
LIN {X 0,Y 512.314,Z 933.181,A -85,B 0,C 180,E1 22625.77,E2 22625.77} C_VEL
LIN {X 0,Y 507.312,Z 953.885,A -85,B 0,C 180,E1 22623.36,E2 22623.36} C_VEL
LIN {X 0,Y 503.709,Z 968.997,A -85,B 0,C 180,E1 22621.338,E2 22621.338} C_VEL
LIN {X 0,Y 500.225,Z 984.121,A -85,B 0,C 180,E1 22619.06,E2 22619.06} C_VEL
LIN {X 0,Y 496.822,Z 999.4,A -85,B 0,C 180,E1 22616.409,E2 22616.409} C_VEL
LIN {X 0,Y 494.45,Z 1010.992,A -85,B 0,C 180,E1 22614.11,E2 22614.11} C_VEL
LIN {X 0,Y 492.342,Z 1022.41,A -85,B 0,C 180,E1 22611.542,E2 22611.542} C_VEL
LIN {X 0,Y 490.518,Z 1033.766,A -85,B 0,C 180,E1 22608.542,E2 22608.542} C_VEL
LIN {X 0,Y 489.479,Z 1041.512,A -85,B 0,C 180,E1 22606.13,E2 22606.13} C_VEL
LIN {X 0,Y 488.753,Z 1048.4,A -85,B 0,C 180,E1 22603.607,E2 22603.607} C_VEL
LIN {X 0,Y 488.231,Z 1055.141,A -85,B 0,C 180,E1 22600.568,E2 22600.568} C_VEL
LIN {X 0,Y 488.015,Z 1059.709,A -85,B 0,C 180,E1 22597.772,E2 22597.772} C_VEL
LIN {X 0,Y 487.923,Z 1062.512,A -85,B 0,C 180,E1 22595.409,E2 22595.409} C_VEL
LIN {X 0,Y 487.913,Z 1064.38,A -85,B 0,C 180,E1 22592.937,E2 22592.937} C_VEL
LIN {X 0,Y 487.914,Z 1065.247,A -85,B 0,C 180,E1 22590,E2 22590} C_VEL
LIN {X 0,Y 487.914,Z 1064.449,A -85,B 0,C 180,E1 22587.181,E2 22587.181} C_VEL
LIN {X 0,Y 487.923,Z 1062.628,A -85,B 0,C 180,E1 22584.709,E2 22584.709} C_VEL
LIN {X 0,Y 488.007,Z 1059.872,A -85,B 0,C 180,E1 22582.347,E2 22582.347} C_VEL
LIN {X 0,Y 488.187,Z 1055.678,A -85,B 0,C 180,E1 22579.736,E2 22579.736} C_VEL
LIN {X 0,Y 488.696,Z 1049.017,A -85,B 0,C 180,E1 22576.632,E2 22576.632} C_VEL
LIN {X 0,Y 489.402,Z 1042.232,A -85,B 0,C 180,E1 22574.111,E2 22574.111} C_VEL
LIN {X 0,Y 490.398,Z 1034.595,A -85,B 0,C 180,E1 22571.7,E2 22571.7} C_VEL
LIN {X 0,Y 492.117,Z 1023.864,A -85,B 0,C 180,E1 22568.798,E2 22568.798} C_VEL
LIN {X 0,Y 494.215,Z 1012.093,A -85,B 0,C 180,E1 22566.132,E2 22566.132} C_VEL
LIN {X 0,Y 496.535,Z 1000.531,A -85,B 0,C 180,E1 22563.832,E2 22563.832} C_VEL
LIN {X 0,Y 499.838,Z 985.334,A -85,B 0,C 180,E1 22561.177,E2 22561.177} C_VEL
LIN {X 0,Y 503.431,Z 969.303,A -85,B 0,C 180,E1 22558.776,E2 22558.776} C_VEL
LIN {X 0,Y 506.97,Z 954.009,A -85,B 0,C 180,E1 22556.747,E2 22556.747} C_VEL
LIN {X 0,Y 511.779,Z 933.399,A -85,B 0,C 180,E1 22554.367,E2 22554.367} C_VEL
LIN {X 0,Y 515.726,Z 916.156,A -85,B 0,C 180,E1 22552.639,E2 22552.639} C_VEL
LIN {X 0,Y 519.907,Z 897.501,A -85,B 0,C 180,E1 22550.985,E2 22550.985} C_VEL
LIN {X 0,Y 524.698,Z 874.894,A -85,B 0,C 180,E1 22549.256,E2 22549.256} C_VEL
LIN {X 0,Y 528.468,Z 855.855,A -85,B 0,C 180,E1 22548,E2 22548} C_VEL
LIN {X 0,Y 531.985,Z 836.859,A -85,B 0,C 180,E1 22546.905,E2 22546.905} C_VEL
LIN {X 0,Y 535.935,Z 813.568,A -85,B 0,C 180,E1 22545.752,E2 22545.752} C_VEL
LIN {X 0,Y 539.25,Z 790.544,A -85,B 0,C 180,E1 22544.82,E2 22544.82} C_VEL
LIN {X 0,Y 541.763,Z 770.624,A -85,B 0,C 180,E1 22544.148,E2 22544.148} C_VEL
LIN {X 0,Y 544.086,Z 748.705,A -85,B 0,C 180,E1 22543.546,E2 22543.546} C_VEL
LIN {X 0,Y 546.312,Z 720.51,A -85,B 0,C 180,E1 22542.974,E2 22542.974} C_VEL
LIN {X 0,Y 549.972,Z 626.641,A -85,B 0,C 180,E1 22541.583,E2 22541.583} C_VEL
LIN {X 0,Y 558.827,Z 398.138,A -85,B 0,C 180,E1 22538.222,E2 22538.222} C_VEL
LIN {X 0,Y 559.345,Z 382.213,A -85,B 0,C 180,E1 22537.97,E2 22537.97} C_VEL
LIN {X 0,Y 546.036,Z 360.84,A -85,B 0,C 180,E1 22535.778,E2 22535.778} C_VEL
LIN {X 0,Y 534.383,Z 343.246,A -85,B 0,C 180,E1 22533.696,E2 22533.696} C_VEL
LIN {X 0,Y 523.153,Z 327.48,A -85,B 0,C 180,E1 22531.516,E2 22531.516} C_VEL
LIN {X 0,Y 515.346,Z 317.151,A -85,B 0,C 180,E1 22529.878,E2 22529.878} C_VEL
LIN {X 0,Y 511.418,Z 311.952,A -85,B 0,C 180,E1 22529.004,E2 22529.004} C_VEL
LIN {X 0,Y 504.478,Z 303.097,A -85,B 0,C 180,E1 22527.376,E2 22527.376} C_VEL
LIN {X 0,Y 501.32,Z 299.391,A -85,B 0,C 180,E1 22526.601,E2 22526.601} C_VEL
LIN {X 0,Y 499.898,Z 297.474,A -85,B 0,C 180,E1 22526.234,E2 22526.234} C_VEL
LIN {X 0,Y 496.782,Z 294.58,A -85,B 0,C 180,E1 22525.45,E2 22525.45} C_VEL
LIN {X 0,Y 494.893,Z 291.407,A -85,B 0,C 180,E1 22524.914,E2 22524.914} C_VEL
LIN {X 0,Y 491.643,Z 288.962,A -85,B 0,C 180,E1 22524.059,E2 22524.059} C_VEL
LIN {X 0,Y 490.029,Z 285.526,A -85,B 0,C 180,E1 22523.447,E2 22523.447} C_VEL
LIN {X 0,Y 489.974,Z 284.938,A -85,B 0,C 180,E1 22522.941,E2 22522.941} C_VEL
LIN {X 0,Y 489.929,Z 284.932,A -85,B 0,C 180,E1 22519.459,E2 22519.459} C_VEL
LIN {X 0,Y 489.928,Z 284.929,A -85,B 0,C 180,E1 22515.872,E2 22515.872} C_VEL
LIN {X 0,Y 489.979,Z 284.918,A -85,B 0,C 180,E1 22512.493,E2 22512.493} C_VEL
LIN {X 0,Y 489.939,Z 284.926,A -85,B 0,C 180,E1 22509.041,E2 22509.041} C_VEL
LIN {X 0,Y 489.926,Z 284.943,A -85,B 0,C 180,E1 22505.622,E2 22505.622} C_VEL
LIN {X 0,Y 489.973,Z 284.947,A -85,B 0,C 180,E1 22502.222,E2 22502.222} C_VEL
LIN {X 0,Y 489.941,Z 284.931,A -85,B 0,C 180,E1 22498.831,E2 22498.831} C_VEL
LIN {X 0,Y 489.921,Z 284.923,A -85,B 0,C 180,E1 22495.317,E2 22495.317} C_VEL
LIN {X 0,Y 489.959,Z 284.921,A -85,B 0,C 180,E1 22491.905,E2 22491.905} C_VEL
LIN {X 0,Y 489.97,Z 284.932,A -85,B 0,C 180,E1 22488.344,E2 22488.344} C_VEL
LIN {X 0,Y 489.926,Z 284.955,A -85,B 0,C 180,E1 22484.978,E2 22484.978} C_VEL
LIN {X 0,Y 489.938,Z 284.944,A -85,B 0,C 180,E1 22481.435,E2 22481.435} C_VEL
LIN {X 0,Y 489.991,Z 284.928,A -85,B 0,C 180,E1 22477.946,E2 22477.946} C_VEL
LIN {X 0,Y 489.931,Z 284.847,A -85,B 0,C 180,E1 22474.43,E2 22474.43} C_VEL
LIN {X 0,Y 490.003,Z 285.289,A -85,B 0,C 180,E1 22473.456,E2 22473.456} C_VEL
LIN {X 0,Y 490.54,Z 287.097,A -85,B 0,C 180,E1 22473.095,E2 22473.095} C_VEL
LIN {X 0,Y 492.526,Z 289.822,A -85,B 0,C 180,E1 22472.518,E2 22472.518} C_VEL
LIN {X 0,Y 495.315,Z 291.797,A -85,B 0,C 180,E1 22471.795,E2 22471.795} C_VEL
LIN {X 0,Y 497.45,Z 295.407,A -85,B 0,C 180,E1 22471.193,E2 22471.193} C_VEL
LIN {X 0,Y 500.728,Z 298.318,A -85,B 0,C 180,E1 22470.381,E2 22470.381} C_VEL
LIN {X 0,Y 503.507,Z 302.224,A -85,B 0,C 180,E1 22469.675,E2 22469.675} C_VEL
LIN {X 0,Y 505.923,Z 304.469,A -85,B 0,C 180,E1 22469.112,E2 22469.112} C_VEL
LIN {X 0,Y 509.404,Z 308.869,A -85,B 0,C 180,E1 22468.294,E2 22468.294} C_VEL
LIN {X 0,Y 511.078,Z 310.86,A -85,B 0,C 180,E1 22467.915,E2 22467.915} C_VEL
LIN {X 0,Y 515.919,Z 316.858,A -85,B 0,C 180,E1 22466.85,E2 22466.85} C_VEL
LIN {X 0,Y 521.003,Z 323.237,A -85,B 0,C 180,E1 22465.784,E2 22465.784} C_VEL
LIN {X 0,Y 529.763,Z 334.442,A -85,B 0,C 180,E1 22464.056,E2 22464.056} C_VEL
LIN {X 0,Y 540.734,Z 350.206,A -85,B 0,C 180,E1 22462.026,E2 22462.026} C_VEL
LIN {X 0,Y 551.436,Z 366.612,A -85,B 0,C 180,E1 22460.185,E2 22460.185} C_VEL
LIN {X 0,Y 559.415,Z 379.479,A -85,B 0,C 180,E1 22458.892,E2 22458.892} C_VEL
LIN {X 0,Y 551.367,Z 586.373,A -85,B 0,C 180,E1 22455.84,E2 22455.84} C_VEL
LIN {X 0,Y 546.483,Z 712.586,A -85,B 0,C 180,E1 22453.976,E2 22453.976} C_VEL
LIN {X 0,Y 544.401,Z 739.902,A -85,B 0,C 180,E1 22453.427,E2 22453.427} C_VEL
LIN {X 0,Y 542.007,Z 762.848,A -85,B 0,C 180,E1 22452.796,E2 22452.796} C_VEL
LIN {X 0,Y 539.47,Z 783.237,A -85,B 0,C 180,E1 22452.105,E2 22452.105} C_VEL
LIN {X 0,Y 535.995,Z 807.343,A -85,B 0,C 180,E1 22451.115,E2 22451.115} C_VEL
LIN {X 0,Y 532.157,Z 829.898,A -85,B 0,C 180,E1 22449.985,E2 22449.985} C_VEL
LIN {X 0,Y 528.69,Z 848.643,A -85,B 0,C 180,E1 22448.895,E2 22448.895} C_VEL
LIN {X 0,Y 524.607,Z 869.224,A -85,B 0,C 180,E1 22447.521,E2 22447.521} C_VEL
LIN {X 0,Y 522.713,Z 877.924,A -85,B 0,C 180,E1 22446.871,E2 22446.871} C_VEL
LIN {X 0,Y 520.546,Z 884.408,A -85,B 0,C 180,E1 22446.443,E2 22446.443} C_VEL
LIN {X 0,Y 511.726,Z 901.358,A -85,B 0,C 180,E1 22445.437,E2 22445.437} C_VEL
LIN {X 0,Y 509.869,Z 906.435,A -85,B 0,C 180,E1 22445.007,E2 22445.007} C_VEL
LIN {X 0,Y 505.862,Z 923.1,A -85,B 0,C 180,E1 22443.332,E2 22443.332} C_VEL
LIN {X 0,Y 501.363,Z 941.565,A -85,B 0,C 180,E1 22441.233,E2 22441.233} C_VEL
LIN {X 0,Y 497.076,Z 958.813,A -85,B 0,C 180,E1 22438.952,E2 22438.952} C_VEL
LIN {X 0,Y 493.686,Z 972.848,A -85,B 0,C 180,E1 22436.85,E2 22436.85} C_VEL
LIN {X 0,Y 490.075,Z 988.379,A -85,B 0,C 180,E1 22434.211,E2 22434.211} C_VEL
LIN {X 0,Y 487.133,Z 1001.692,A -85,B 0,C 180,E1 22431.556,E2 22431.556} C_VEL
LIN {X 0,Y 484.986,Z 1012.339,A -85,B 0,C 180,E1 22429.136,E2 22429.136} C_VEL
LIN {X 0,Y 482.987,Z 1023.684,A -85,B 0,C 180,E1 22426.14,E2 22426.14} C_VEL
LIN {X 0,Y 481.701,Z 1032.182,A -85,B 0,C 180,E1 22423.443,E2 22423.443} C_VEL
LIN {X 0,Y 480.908,Z 1038.946,A -85,B 0,C 180,E1 22420.906,E2 22420.906} C_VEL
LIN {X 0,Y 480.323,Z 1045.539,A -85,B 0,C 180,E1 22417.897,E2 22417.897} C_VEL
LIN {X 0,Y 480.034,Z 1050.322,A -85,B 0,C 180,E1 22414.899,E2 22414.899} C_VEL
LIN {X 0,Y 479.929,Z 1053.088,A -85,B 0,C 180,E1 22412.508,E2 22412.508} C_VEL
LIN {X 0,Y 479.93,Z 1054.943,A -85,B 0,C 180,E1 22410,E2 22410} C_VEL
LIN {X 0,Y 479.901,Z 1055.805,A -85,B 0,C 180,E1 22407.134,E2 22407.134} C_VEL
LIN {X 0,Y 479.918,Z 1055.075,A -85,B 0,C 180,E1 22404.14,E2 22404.14} C_VEL
LIN {X 0,Y 479.933,Z 1053.291,A -85,B 0,C 180,E1 22401.614,E2 22401.614} C_VEL
LIN {X 0,Y 480.025,Z 1050.57,A -85,B 0,C 180,E1 22399.195,E2 22399.195} C_VEL
LIN {X 0,Y 480.246,Z 1046.357,A -85,B 0,C 180,E1 22396.487,E2 22396.487} C_VEL
LIN {X 0,Y 480.818,Z 1039.746,A -85,B 0,C 180,E1 22393.323,E2 22393.323} C_VEL
LIN {X 0,Y 481.606,Z 1032.939,A -85,B 0,C 180,E1 22390.725,E2 22390.725} C_VEL
LIN {X 0,Y 482.739,Z 1025.255,A -85,B 0,C 180,E1 22388.238,E2 22388.238} C_VEL
LIN {X 0,Y 484.691,Z 1014.173,A -85,B 0,C 180,E1 22385.19,E2 22385.19} C_VEL
LIN {X 0,Y 487.033,Z 1002.517,A -85,B 0,C 180,E1 22382.488,E2 22382.488} C_VEL
LIN {X 0,Y 489.764,Z 990.214,A -85,B 0,C 180,E1 22379.988,E2 22379.988} C_VEL
LIN {X 0,Y 493.564,Z 974.411,A -85,B 0,C 180,E1 22377.218,E2 22377.218} C_VEL
LIN {X 0,Y 497.121,Z 960.052,A -85,B 0,C 180,E1 22375.024,E2 22375.024} C_VEL
LIN {X 0,Y 501.555,Z 942.794,A -85,B 0,C 180,E1 22372.696,E2 22372.696} C_VEL
LIN {X 0,Y 506.335,Z 923.964,A -85,B 0,C 180,E1 22370.515,E2 22370.515} C_VEL
LIN {X 0,Y 510.445,Z 907.545,A -85,B 0,C 180,E1 22368.839,E2 22368.839} C_VEL
LIN {X 0,Y 515.265,Z 887.878,A -85,B 0,C 180,E1 22367.068,E2 22367.068} C_VEL
LIN {X 0,Y 520.272,Z 865.891,A -85,B 0,C 180,E1 22365.377,E2 22365.377} C_VEL
LIN {X 0,Y 524.353,Z 846.847,A -85,B 0,C 180,E1 22364.109,E2 22364.109} C_VEL
LIN {X 0,Y 528.448,Z 826.352,A -85,B 0,C 180,E1 22362.925,E2 22362.925} C_VEL
LIN {X 0,Y 532.819,Z 801.456,A -85,B 0,C 180,E1 22361.719,E2 22361.719} C_VEL
LIN {X 0,Y 535.928,Z 781.296,A -85,B 0,C 180,E1 22360.91,E2 22360.91} C_VEL
LIN {X 0,Y 538.613,Z 761.206,A -85,B 0,C 180,E1 22360.235,E2 22360.235} C_VEL
LIN {X 0,Y 541.424,Z 735.969,A -85,B 0,C 180,E1 22359.558,E2 22359.558} C_VEL
LIN {X 0,Y 543.33,Z 710.858,A -85,B 0,C 180,E1 22359.07,E2 22359.07} C_VEL
LIN {X 0,Y 553.175,Z 483.303,A -85,B 0,C 180,E1 22355.666,E2 22355.666} C_VEL
LIN {X 0,Y 557.475,Z 384.023,A -85,B 0,C 180,E1 22354.153,E2 22354.153} C_VEL
LIN {X 0,Y 545.09,Z 364.705,A -85,B 0,C 180,E1 22351.863,E2 22351.863} C_VEL
LIN {X 0,Y 532.773,Z 346.982,A -85,B 0,C 180,E1 22349.361,E2 22349.361} C_VEL
LIN {X 0,Y 523.584,Z 334.916,A -85,B 0,C 180,E1 22347.31,E2 22347.31} C_VEL
LIN {X 0,Y 517.932,Z 328.167,A -85,B 0,C 180,E1 22345.961,E2 22345.961} C_VEL
LIN {X 0,Y 513.635,Z 322.845,A -85,B 0,C 180,E1 22344.865,E2 22344.865} C_VEL
LIN {X 0,Y 509.891,Z 318.114,A -85,B 0,C 180,E1 22343.857,E2 22343.857} C_VEL
LIN {X 0,Y 505.942,Z 313.912,A -85,B 0,C 180,E1 22342.759,E2 22342.759} C_VEL
LIN {X 0,Y 504.444,Z 311.815,A -85,B 0,C 180,E1 22342.308,E2 22342.308} C_VEL
LIN {X 0,Y 501.053,Z 308.495,A -85,B 0,C 180,E1 22341.297,E2 22341.297} C_VEL
LIN {X 0,Y 499.09,Z 305.553,A -85,B 0,C 180,E1 22340.647,E2 22340.647} C_VEL
LIN {X 0,Y 495.812,Z 302.722,A -85,B 0,C 180,E1 22339.589,E2 22339.589} C_VEL
LIN {X 0,Y 493.643,Z 299.27,A -85,B 0,C 180,E1 22338.788,E2 22338.788} C_VEL
LIN {X 0,Y 490.218,Z 296.76,A -85,B 0,C 180,E1 22337.57,E2 22337.57} C_VEL
LIN {X 0,Y 488.263,Z 293.581,A -85,B 0,C 180,E1 22336.752,E2 22336.752} C_VEL
LIN {X 0,Y 487.521,Z 292.621,A -85,B 0,C 180,E1 22336.441,E2 22336.441} C_VEL
LIN {X 0,Y 483.953,Z 290.21,A -85,B 0,C 180,E1 22334.967,E2 22334.967} C_VEL
LIN {X 0,Y 482.334,Z 287.288,A -85,B 0,C 180,E1 22334.129,E2 22334.129} C_VEL
LIN {X 0,Y 482.051,Z 286.133,A -85,B 0,C 180,E1 22333.556,E2 22333.556} C_VEL
LIN {X 0,Y 481.995,Z 285.939,A -85,B 0,C 180,E1 22330.486,E2 22330.486} C_VEL
LIN {X 0,Y 481.976,Z 285.844,A -85,B 0,C 180,E1 22326.911,E2 22326.911} C_VEL
LIN {X 0,Y 482.025,Z 285.937,A -85,B 0,C 180,E1 22323.449,E2 22323.449} C_VEL
LIN {X 0,Y 482.019,Z 285.838,A -85,B 0,C 180,E1 22319.881,E2 22319.881} C_VEL
LIN {X 0,Y 481.991,Z 285.945,A -85,B 0,C 180,E1 22316.432,E2 22316.432} C_VEL
LIN {X 0,Y 481.977,Z 285.842,A -85,B 0,C 180,E1 22312.73,E2 22312.73} C_VEL
LIN {X 0,Y 482.027,Z 285.923,A -85,B 0,C 180,E1 22309.24,E2 22309.24} C_VEL
LIN {X 0,Y 482.013,Z 285.84,A -85,B 0,C 180,E1 22305.708,E2 22305.708} C_VEL
LIN {X 0,Y 482.075,Z 286.165,A -85,B 0,C 180,E1 22303.491,E2 22303.491} C_VEL
LIN {X 0,Y 482.355,Z 287.457,A -85,B 0,C 180,E1 22302.943,E2 22302.943} C_VEL
LIN {X 0,Y 483.938,Z 290.22,A -85,B 0,C 180,E1 22302.132,E2 22302.132} C_VEL
LIN {X 0,Y 488.146,Z 293.218,A -85,B 0,C 180,E1 22300.402,E2 22300.402} C_VEL
LIN {X 0,Y 490.081,Z 296.545,A -85,B 0,C 180,E1 22299.581,E2 22299.581} C_VEL
LIN {X 0,Y 493.158,Z 299.003,A -85,B 0,C 180,E1 22298.47,E2 22298.47} C_VEL
LIN {X 0,Y 494.027,Z 299.759,A -85,B 0,C 180,E1 22298.167,E2 22298.167} C_VEL
LIN {X 0,Y 496.399,Z 303.494,A -85,B 0,C 180,E1 22297.3,E2 22297.3} C_VEL
LIN {X 0,Y 499.6,Z 306.205,A -85,B 0,C 180,E1 22296.279,E2 22296.279} C_VEL
LIN {X 0,Y 502.463,Z 310.184,A -85,B 0,C 180,E1 22295.361,E2 22295.361} C_VEL
LIN {X 0,Y 505.091,Z 312.813,A -85,B 0,C 180,E1 22294.59,E2 22294.59} C_VEL
LIN {X 0,Y 512.965,Z 322.664,A -85,B 0,C 180,E1 22292.391,E2 22292.391} C_VEL
LIN {X 0,Y 518.849,Z 330.388,A -85,B 0,C 180,E1 22290.882,E2 22290.882} C_VEL
LIN {X 0,Y 526.012,Z 339.806,A -85,B 0,C 180,E1 22289.183,E2 22289.183} C_VEL
LIN {X 0,Y 536.243,Z 354.22,A -85,B 0,C 180,E1 22286.948,E2 22286.948} C_VEL
LIN {X 0,Y 546.474,Z 369.508,A -85,B 0,C 180,E1 22284.901,E2 22284.901} C_VEL
LIN {X 0,Y 556.708,Z 385.767,A -85,B 0,C 180,E1 22283.009,E2 22283.009} C_VEL
LIN {X 0,Y 557.582,Z 387.562,A -85,B 0,C 180,E1 22282.846,E2 22282.846} C_VEL
LIN {X 0,Y 547.423,Z 619.267,A -85,B 0,C 180,E1 22279.384,E2 22279.384} C_VEL
LIN {X 0,Y 543.044,Z 720.177,A -85,B 0,C 180,E1 22277.865,E2 22277.865} C_VEL
LIN {X 0,Y 540.683,Z 748.115,A -85,B 0,C 180,E1 22277.296,E2 22277.296} C_VEL
LIN {X 0,Y 538.191,Z 769.856,A -85,B 0,C 180,E1 22276.699,E2 22276.699} C_VEL
LIN {X 0,Y 535.492,Z 789.658,A -85,B 0,C 180,E1 22276.032,E2 22276.032} C_VEL
LIN {X 0,Y 531.795,Z 813.417,A -85,B 0,C 180,E1 22275.064,E2 22275.064} C_VEL
LIN {X 0,Y 527.584,Z 836.351,A -85,B 0,C 180,E1 22273.92,E2 22273.92} C_VEL
LIN {X 0,Y 523.767,Z 855.377,A -85,B 0,C 180,E1 22272.813,E2 22272.813} C_VEL
LIN {X 0,Y 519.453,Z 875.525,A -85,B 0,C 180,E1 22271.465,E2 22271.465} C_VEL
LIN {X 0,Y 514.083,Z 898.788,A -85,B 0,C 180,E1 22269.64,E2 22269.64} C_VEL
LIN {X 0,Y 509.897,Z 916.046,A -85,B 0,C 180,E1 22268.077,E2 22268.077} C_VEL
LIN {X 0,Y 505.632,Z 933.261,A -85,B 0,C 180,E1 22266.318,E2 22266.318} C_VEL
LIN {X 0,Y 500.395,Z 953.932,A -85,B 0,C 180,E1 22263.883,E2 22263.883} C_VEL
LIN {X 0,Y 496.588,Z 969.148,A -85,B 0,C 180,E1 22261.82,E2 22261.82} C_VEL
LIN {X 0,Y 492.792,Z 984.904,A -85,B 0,C 180,E1 22259.408,E2 22259.408} C_VEL
LIN {X 0,Y 489.231,Z 1000.023,A -85,B 0,C 180,E1 22256.72,E2 22256.72} C_VEL
LIN {X 0,Y 486.758,Z 1011.538,A -85,B 0,C 180,E1 22254.386,E2 22254.386} C_VEL
LIN {X 0,Y 484.394,Z 1023.809,A -85,B 0,C 180,E1 22251.557,E2 22251.557} C_VEL
LIN {X 0,Y 482.57,Z 1034.51,A -85,B 0,C 180,E1 22248.608,E2 22248.608} C_VEL
LIN {X 0,Y 481.502,Z 1042.143,A -85,B 0,C 180,E1 22246.157,E2 22246.157} C_VEL
LIN {X 0,Y 480.699,Z 1049.539,A -85,B 0,C 180,E1 22243.349,E2 22243.349} C_VEL
LIN {X 0,Y 480.194,Z 1055.801,A -85,B 0,C 180,E1 22240.316,E2 22240.316} C_VEL
LIN {X 0,Y 480.016,Z 1059.791,A -85,B 0,C 180,E1 22237.782,E2 22237.782} C_VEL
LIN {X 0,Y 479.923,Z 1062.548,A -85,B 0,C 180,E1 22235.38,E2 22235.38} C_VEL
LIN {X 0,Y 479.914,Z 1064.439,A -85,B 0,C 180,E1 22232.747,E2 22232.747} C_VEL
LIN {X 0,Y 479.902,Z 1065.108,A -85,B 0,C 180,E1 22229.642,E2 22229.642} C_VEL
LIN {X 0,Y 479.913,Z 1064.302,A -85,B 0,C 180,E1 22227.014,E2 22227.014} C_VEL
LIN {X 0,Y 479.922,Z 1062.435,A -85,B 0,C 180,E1 22224.501,E2 22224.501} C_VEL
LIN {X 0,Y 480.023,Z 1059.633,A -85,B 0,C 180,E1 22222.098,E2 22222.098} C_VEL
LIN {X 0,Y 480.281,Z 1054.763,A -85,B 0,C 180,E1 22219.079,E2 22219.079} C_VEL
LIN {X 0,Y 480.852,Z 1048.023,A -85,B 0,C 180,E1 22216.042,E2 22216.042} C_VEL
LIN {X 0,Y 481.638,Z 1041.085,A -85,B 0,C 180,E1 22213.476,E2 22213.476} C_VEL
LIN {X 0,Y 483.041,Z 1031.638,A -85,B 0,C 180,E1 22210.533,E2 22210.533} C_VEL
LIN {X 0,Y 484.926,Z 1020.638,A -85,B 0,C 180,E1 22207.704,E2 22207.704} C_VEL
LIN {X 0,Y 486.974,Z 1010.226,A -85,B 0,C 180,E1 22205.367,E2 22205.367} C_VEL
LIN {X 0,Y 489.944,Z 996.533,A -85,B 0,C 180,E1 22202.666,E2 22202.666} C_VEL
LIN {X 0,Y 493.412,Z 981.271,A -85,B 0,C 180,E1 22200.099,E2 22200.099} C_VEL
LIN {X 0,Y 496.703,Z 967.405,A -85,B 0,C 180,E1 22198.033,E2 22198.033} C_VEL
LIN {X 0,Y 501.026,Z 949.783,A -85,B 0,C 180,E1 22195.712,E2 22195.712} C_VEL
LIN {X 0,Y 505.515,Z 931.131,A -85,B 0,C 180,E1 22193.602,E2 22193.602} C_VEL
LIN {X 0,Y 509.437,Z 914.666,A -85,B 0,C 180,E1 22191.954,E2 22191.954} C_VEL
LIN {X 0,Y 514.187,Z 894.282,A -85,B 0,C 180,E1 22190.153,E2 22190.153} C_VEL
LIN {X 0,Y 518.793,Z 872.923,A -85,B 0,C 180,E1 22188.545,E2 22188.545} C_VEL
LIN {X 0,Y 522.799,Z 853.31,A -85,B 0,C 180,E1 22187.259,E2 22187.259} C_VEL
LIN {X 0,Y 527.161,Z 830.322,A -85,B 0,C 180,E1 22185.961,E2 22185.961} C_VEL
LIN {X 0,Y 531.048,Z 806.584,A -85,B 0,C 180,E1 22184.855,E2 22184.855} C_VEL
LIN {X 0,Y 534.12,Z 785.653,A -85,B 0,C 180,E1 22184.04,E2 22184.04} C_VEL
LIN {X 0,Y 537.252,Z 760.599,A -85,B 0,C 180,E1 22183.244,E2 22183.244} C_VEL
LIN {X 0,Y 539.618,Z 735.875,A -85,B 0,C 180,E1 22182.655,E2 22182.655} C_VEL
LIN {X 0,Y 541.127,Z 713.573,A -85,B 0,C 180,E1 22182.251,E2 22182.251} C_VEL
LIN {X 0,Y 550.46,Z 478.084,A -85,B 0,C 180,E1 22178.768,E2 22178.768} C_VEL
LIN {X 0,Y 554.18,Z 386.014,A -85,B 0,C 180,E1 22177.39,E2 22177.39} C_VEL
LIN {X 0,Y 541.753,Z 365.983,A -85,B 0,C 180,E1 22175.288,E2 22175.288} C_VEL
LIN {X 0,Y 530.761,Z 349.302,A -85,B 0,C 180,E1 22173.277,E2 22173.277} C_VEL
LIN {X 0,Y 519.916,Z 333.875,A -85,B 0,C 180,E1 22171.122,E2 22171.122} C_VEL
LIN {X 0,Y 512.194,Z 323.563,A -85,B 0,C 180,E1 22169.464,E2 22169.464} C_VEL
LIN {X 0,Y 508.554,Z 318.697,A -85,B 0,C 180,E1 22168.636,E2 22168.636} C_VEL
LIN {X 0,Y 501.804,Z 310.065,A -85,B 0,C 180,E1 22167.021,E2 22167.021} C_VEL
LIN {X 0,Y 498.404,Z 305.783,A -85,B 0,C 180,E1 22166.159,E2 22166.159} C_VEL
LIN {X 0,Y 497.058,Z 304.423,A -85,B 0,C 180,E1 22165.818,E2 22165.818} C_VEL
LIN {X 0,Y 493.934,Z 301.016,A -85,B 0,C 180,E1 22164.998,E2 22164.998} C_VEL
LIN {X 0,Y 492.527,Z 298.75,A -85,B 0,C 180,E1 22164.593,E2 22164.593} C_VEL
LIN {X 0,Y 489.269,Z 295.995,A -85,B 0,C 180,E1 22163.709,E2 22163.709} C_VEL
LIN {X 0,Y 487.247,Z 292.492,A -85,B 0,C 180,E1 22163.076,E2 22163.076} C_VEL
LIN {X 0,Y 483.846,Z 290.14,A -85,B 0,C 180,E1 22162.093,E2 22162.093} C_VEL
LIN {X 0,Y 482.111,Z 286.601,A -85,B 0,C 180,E1 22161.376,E2 22161.376} C_VEL
LIN {X 0,Y 482.035,Z 285.946,A -85,B 0,C 180,E1 22160.903,E2 22160.903} C_VEL
LIN {X 0,Y 481.991,Z 285.921,A -85,B 0,C 180,E1 22157.381,E2 22157.381} C_VEL
LIN {X 0,Y 481.989,Z 285.928,A -85,B 0,C 180,E1 22153.802,E2 22153.802} C_VEL
LIN {X 0,Y 482.038,Z 285.938,A -85,B 0,C 180,E1 22150.397,E2 22150.397} C_VEL
LIN {X 0,Y 482.008,Z 285.928,A -85,B 0,C 180,E1 22146.91,E2 22146.91} C_VEL
LIN {X 0,Y 481.984,Z 285.916,A -85,B 0,C 180,E1 22143.449,E2 22143.449} C_VEL
LIN {X 0,Y 482.014,Z 285.907,A -85,B 0,C 180,E1 22140,E2 22140} C_VEL
LIN {X 0,Y 482.022,Z 285.915,A -85,B 0,C 180,E1 22136.551,E2 22136.551} C_VEL
LIN {X 0,Y 481.986,Z 285.94,A -85,B 0,C 180,E1 22133.089,E2 22133.089} C_VEL
LIN {X 0,Y 481.993,Z 285.938,A -85,B 0,C 180,E1 22129.481,E2 22129.481} C_VEL
LIN {X 0,Y 482.034,Z 285.917,A -85,B 0,C 180,E1 22125.954,E2 22125.954} C_VEL
LIN {X 0,Y 482.007,Z 285.912,A -85,B 0,C 180,E1 22122.495,E2 22122.495} C_VEL
LIN {X 0,Y 481.985,Z 285.913,A -85,B 0,C 180,E1 22118.968,E2 22118.968} C_VEL
LIN {X 0,Y 482.05,Z 286.11,A -85,B 0,C 180,E1 22115.658,E2 22115.658} C_VEL
LIN {X 0,Y 482.358,Z 287.471,A -85,B 0,C 180,E1 22115.245,E2 22115.245} C_VEL
LIN {X 0,Y 483.996,Z 290.234,A -85,B 0,C 180,E1 22114.682,E2 22114.682} C_VEL
LIN {X 0,Y 487.581,Z 292.934,A -85,B 0,C 180,E1 22113.642,E2 22113.642} C_VEL
LIN {X 0,Y 489.725,Z 296.489,A -85,B 0,C 180,E1 22112.981,E2 22112.981} C_VEL
LIN {X 0,Y 493.003,Z 299.308,A -85,B 0,C 180,E1 22112.095,E2 22112.095} C_VEL
LIN {X 0,Y 495.709,Z 303.237,A -85,B 0,C 180,E1 22111.343,E2 22111.343} C_VEL
LIN {X 0,Y 498.316,Z 305.628,A -85,B 0,C 180,E1 22110.686,E2 22110.686} C_VEL
LIN {X 0,Y 501.51,Z 309.808,A -85,B 0,C 180,E1 22109.872,E2 22109.872} C_VEL
LIN {X 0,Y 503.563,Z 311.897,A -85,B 0,C 180,E1 22109.382,E2 22109.382} C_VEL
LIN {X 0,Y 507.367,Z 316.447,A -85,B 0,C 180,E1 22108.484,E2 22108.484} C_VEL
LIN {X 0,Y 513.517,Z 324.306,A -85,B 0,C 180,E1 22107.094,E2 22107.094} C_VEL
LIN {X 0,Y 521.021,Z 333.674,A -85,B 0,C 180,E1 22105.519,E2 22105.519} C_VEL
LIN {X 0,Y 529.171,Z 344.645,A -85,B 0,C 180,E1 22103.909,E2 22103.909} C_VEL
LIN {X 0,Y 541.959,Z 363.611,A -85,B 0,C 180,E1 22101.556,E2 22101.556} C_VEL
LIN {X 0,Y 554.214,Z 383.236,A -85,B 0,C 180,E1 22099.479,E2 22099.479} C_VEL
LIN {X 0,Y 545.874,Z 589.668,A -85,B 0,C 180,E1 22096.415,E2 22096.415} C_VEL
LIN {X 0,Y 540.933,Z 712.651,A -85,B 0,C 180,E1 22094.586,E2 22094.586} C_VEL
LIN {X 0,Y 538.798,Z 739.911,A -85,B 0,C 180,E1 22094.035,E2 22094.035} C_VEL
LIN {X 0,Y 536.327,Z 762.875,A -85,B 0,C 180,E1 22093.402,E2 22093.402} C_VEL
LIN {X 0,Y 533.814,Z 782.48,A -85,B 0,C 180,E1 22092.737,E2 22092.737} C_VEL
LIN {X 0,Y 530.392,Z 805.688,A -85,B 0,C 180,E1 22091.791,E2 22091.791} C_VEL
LIN {X 0,Y 526.23,Z 829.528,A -85,B 0,C 180,E1 22090.6,E2 22090.6} C_VEL
LIN {X 0,Y 522.634,Z 848.326,A -85,B 0,C 180,E1 22089.504,E2 22089.504} C_VEL
LIN {X 0,Y 518.505,Z 868.419,A -85,B 0,C 180,E1 22088.158,E2 22088.158} C_VEL
LIN {X 0,Y 513.42,Z 891.215,A -85,B 0,C 180,E1 22086.371,E2 22086.371} C_VEL
LIN {X 0,Y 509.869,Z 906.435,A -85,B 0,C 180,E1 22085.007,E2 22085.007} C_VEL
LIN {X 0,Y 507.617,Z 912.458,A -85,B 0,C 180,E1 22084.502,E2 22084.502} C_VEL
LIN {X 0,Y 498.51,Z 928.287,A -85,B 0,C 180,E1 22083.28,E2 22083.28} C_VEL
LIN {X 0,Y 496.652,Z 932.999,A -85,B 0,C 180,E1 22082.785,E2 22082.785} C_VEL
LIN {X 0,Y 492.615,Z 948.719,A -85,B 0,C 180,E1 22080.841,E2 22080.841} C_VEL
LIN {X 0,Y 488.526,Z 964.829,A -85,B 0,C 180,E1 22078.591,E2 22078.591} C_VEL
LIN {X 0,Y 484.404,Z 981.14,A -85,B 0,C 180,E1 22075.951,E2 22075.951} C_VEL
LIN {X 0,Y 481.416,Z 993.655,A -85,B 0,C 180,E1 22073.632,E2 22073.632} C_VEL
LIN {X 0,Y 478.46,Z 1007.02,A -85,B 0,C 180,E1 22070.81,E2 22070.81} C_VEL
LIN {X 0,Y 476.157,Z 1018.367,A -85,B 0,C 180,E1 22067.961,E2 22067.961} C_VEL
LIN {X 0,Y 474.676,Z 1026.805,A -85,B 0,C 180,E1 22065.517,E2 22065.517} C_VEL
LIN {X 0,Y 473.424,Z 1035.523,A -85,B 0,C 180,E1 22062.564,E2 22062.564} C_VEL
LIN {X 0,Y 472.591,Z 1042.724,A -85,B 0,C 180,E1 22059.499,E2 22059.499} C_VEL
LIN {X 0,Y 472.189,Z 1047.544,A -85,B 0,C 180,E1 22056.932,E2 22056.932} C_VEL
LIN {X 0,Y 472.009,Z 1051.256,A -85,B 0,C 180,E1 22054.374,E2 22054.374} C_VEL
LIN {X 0,Y 471.915,Z 1054.309,A -85,B 0,C 180,E1 22051.335,E2 22051.335} C_VEL
LIN {X 0,Y 471.899,Z 1055.644,A -85,B 0,C 180,E1 22048.422,E2 22048.422} C_VEL
LIN {X 0,Y 471.905,Z 1055.738,A -85,B 0,C 180,E1 22045.99,E2 22045.99} C_VEL
LIN {X 0,Y 471.916,Z 1054.854,A -85,B 0,C 180,E1 22043.552,E2 22043.552} C_VEL
LIN {X 0,Y 471.945,Z 1052.868,A -85,B 0,C 180,E1 22040.98,E2 22040.98} C_VEL
LIN {X 0,Y 472.108,Z 1049.086,A -85,B 0,C 180,E1 22037.897,E2 22037.897} C_VEL
LIN {X 0,Y 472.478,Z 1044.017,A -85,B 0,C 180,E1 22035.038,E2 22035.038} C_VEL
LIN {X 0,Y 473.089,Z 1038.178,A -85,B 0,C 180,E1 22032.408,E2 22032.408} C_VEL
LIN {X 0,Y 474.154,Z 1030.397,A -85,B 0,C 180,E1 22029.509,E2 22029.509} C_VEL
LIN {X 0,Y 475.823,Z 1020.407,A -85,B 0,C 180,E1 22026.468,E2 22026.468} C_VEL
LIN {X 0,Y 477.76,Z 1010.658,A -85,B 0,C 180,E1 22023.928,E2 22023.928} C_VEL
LIN {X 0,Y 480.654,Z 997.776,A -85,B 0,C 180,E1 22021.007,E2 22021.007} C_VEL
LIN {X 0,Y 483.982,Z 983.9,A -85,B 0,C 180,E1 22018.341,E2 22018.341} C_VEL
LIN {X 0,Y 487.192,Z 971.351,A -85,B 0,C 180,E1 22016.208,E2 22016.208} C_VEL
LIN {X 0,Y 491.635,Z 954.75,A -85,B 0,C 180,E1 22013.713,E2 22013.713} C_VEL
LIN {X 0,Y 496.377,Z 936.825,A -85,B 0,C 180,E1 22011.406,E2 22011.406} C_VEL
LIN {X 0,Y 500.593,Z 920.915,A -85,B 0,C 180,E1 22009.597,E2 22009.597} C_VEL
LIN {X 0,Y 505.778,Z 901.096,A -85,B 0,C 180,E1 22007.613,E2 22007.613} C_VEL
LIN {X 0,Y 510.897,Z 880.229,A -85,B 0,C 180,E1 22005.835,E2 22005.835} C_VEL
LIN {X 0,Y 515.307,Z 861.411,A -85,B 0,C 180,E1 22004.434,E2 22004.434} C_VEL
LIN {X 0,Y 520.39,Z 838.104,A -85,B 0,C 180,E1 22002.941,E2 22002.941} C_VEL
LIN {X 0,Y 524.702,Z 815.871,A -85,B 0,C 180,E1 22001.751,E2 22001.751} C_VEL
LIN {X 0,Y 528.334,Z 794.983,A -85,B 0,C 180,E1 22000.799,E2 22000.799} C_VEL
LIN {X 0,Y 532.359,Z 768.083,A -85,B 0,C 180,E1 21999.803,E2 21999.803} C_VEL
LIN {X 0,Y 535.06,Z 745.549,A -85,B 0,C 180,E1 21999.147,E2 21999.147} C_VEL
LIN {X 0,Y 537.341,Z 722.017,A -85,B 0,C 180,E1 21998.62,E2 21998.62} C_VEL
LIN {X 0,Y 539.299,Z 687.085,A -85,B 0,C 180,E1 21998.052,E2 21998.052} C_VEL
LIN {X 0,Y 549.441,Z 458.852,A -85,B 0,C 180,E1 21994.628,E2 21994.628} C_VEL
LIN {X 0,Y 552.678,Z 388.265,A -85,B 0,C 180,E1 21993.553,E2 21993.553} C_VEL
LIN {X 0,Y 541.442,Z 370.523,A -85,B 0,C 180,E1 21991.415,E2 21991.415} C_VEL
LIN {X 0,Y 529.538,Z 353.251,A -85,B 0,C 180,E1 21988.938,E2 21988.938} C_VEL
LIN {X 0,Y 520.794,Z 341.724,A -85,B 0,C 180,E1 21986.943,E2 21986.943} C_VEL
LIN {X 0,Y 515.021,Z 334.731,A -85,B 0,C 180,E1 21985.531,E2 21985.531} C_VEL
LIN {X 0,Y 511.283,Z 330.002,A -85,B 0,C 180,E1 21984.556,E2 21984.556} C_VEL
LIN {X 0,Y 506.911,Z 324.708,A -85,B 0,C 180,E1 21983.358,E2 21983.358} C_VEL
LIN {X 0,Y 503.181,Z 320.252,A -85,B 0,C 180,E1 21982.275,E2 21982.275} C_VEL
LIN {X 0,Y 501.659,Z 318.664,A -85,B 0,C 180,E1 21981.822,E2 21981.822} C_VEL
LIN {X 0,Y 498.315,Z 314.767,A -85,B 0,C 180,E1 21980.772,E2 21980.772} C_VEL
LIN {X 0,Y 497.102,Z 313.03,A -85,B 0,C 180,E1 21980.364,E2 21980.364} C_VEL
LIN {X 0,Y 493.731,Z 309.867,A -85,B 0,C 180,E1 21979.244,E2 21979.244} C_VEL
LIN {X 0,Y 491.728,Z 306.809,A -85,B 0,C 180,E1 21978.495,E2 21978.495} C_VEL
LIN {X 0,Y 488.235,Z 303.964,A -85,B 0,C 180,E1 21977.213,E2 21977.213} C_VEL
LIN {X 0,Y 485.994,Z 300.362,A -85,B 0,C 180,E1 21976.249,E2 21976.249} C_VEL
LIN {X 0,Y 482.476,Z 297.892,A -85,B 0,C 180,E1 21974.768,E2 21974.768} C_VEL
LIN {X 0,Y 480.608,Z 294.691,A -85,B 0,C 180,E1 21973.812,E2 21973.812} C_VEL
LIN {X 0,Y 479.508,Z 293.557,A -85,B 0,C 180,E1 21973.26,E2 21973.26} C_VEL
LIN {X 0,Y 475.867,Z 291.034,A -85,B 0,C 180,E1 21971.33,E2 21971.33} C_VEL
LIN {X 0,Y 474.338,Z 288.207,A -85,B 0,C 180,E1 21970.261,E2 21970.261} C_VEL
LIN {X 0,Y 474.102,Z 287.091,A -85,B 0,C 180,E1 21969.468,E2 21969.468} C_VEL
LIN {X 0,Y 474.05,Z 286.832,A -85,B 0,C 180,E1 21966.297,E2 21966.297} C_VEL
LIN {X 0,Y 474.045,Z 286.897,A -85,B 0,C 180,E1 21962.781,E2 21962.781} C_VEL
LIN {X 0,Y 474.067,Z 286.831,A -85,B 0,C 180,E1 21959.275,E2 21959.275} C_VEL
LIN {X 0,Y 474.088,Z 286.893,A -85,B 0,C 180,E1 21955.767,E2 21955.767} C_VEL
LIN {X 0,Y 474.04,Z 286.831,A -85,B 0,C 180,E1 21952.364,E2 21952.364} C_VEL
LIN {X 0,Y 474.047,Z 286.885,A -85,B 0,C 180,E1 21948.687,E2 21948.687} C_VEL
LIN {X 0,Y 474.176,Z 287.423,A -85,B 0,C 180,E1 21947.208,E2 21947.208} C_VEL
LIN {X 0,Y 474.686,Z 289.137,A -85,B 0,C 180,E1 21946.54,E2 21946.54} C_VEL
LIN {X 0,Y 476.885,Z 291.98,A -85,B 0,C 180,E1 21945.179,E2 21945.179} C_VEL
LIN {X 0,Y 480.444,Z 294.34,A -85,B 0,C 180,E1 21943.372,E2 21943.372} C_VEL
LIN {X 0,Y 482.103,Z 297.483,A -85,B 0,C 180,E1 21942.498,E2 21942.498} C_VEL
LIN {X 0,Y 485.288,Z 299.976,A -85,B 0,C 180,E1 21941.126,E2 21941.126} C_VEL
LIN {X 0,Y 486.41,Z 300.822,A -85,B 0,C 180,E1 21940.673,E2 21940.673} C_VEL
LIN {X 0,Y 488.684,Z 304.43,A -85,B 0,C 180,E1 21939.707,E2 21939.707} C_VEL
LIN {X 0,Y 492.2,Z 307.382,A -85,B 0,C 180,E1 21938.426,E2 21938.426} C_VEL
LIN {X 0,Y 494.932,Z 311.362,A -85,B 0,C 180,E1 21937.428,E2 21937.428} C_VEL
LIN {X 0,Y 497.703,Z 313.798,A -85,B 0,C 180,E1 21936.529,E2 21936.529} C_VEL
LIN {X 0,Y 500.808,Z 317.911,A -85,B 0,C 180,E1 21935.526,E2 21935.526} C_VEL
LIN {X 0,Y 503.137,Z 320.318,A -85,B 0,C 180,E1 21934.831,E2 21934.831} C_VEL
LIN {X 0,Y 510.732,Z 329.981,A -85,B 0,C 180,E1 21932.671,E2 21932.671} C_VEL
LIN {X 0,Y 518.962,Z 340.747,A -85,B 0,C 180,E1 21930.56,E2 21930.56} C_VEL
LIN {X 0,Y 528.624,Z 354.192,A -85,B 0,C 180,E1 21928.307,E2 21928.307} C_VEL
LIN {X 0,Y 538.839,Z 369.158,A -85,B 0,C 180,E1 21926.141,E2 21926.141} C_VEL
LIN {X 0,Y 549.97,Z 386.681,A -85,B 0,C 180,E1 21923.974,E2 21923.974} C_VEL
LIN {X 0,Y 552.709,Z 391.531,A -85,B 0,C 180,E1 21923.461,E2 21923.461} C_VEL
LIN {X 0,Y 542.229,Z 622.173,A -85,B 0,C 180,E1 21919.995,E2 21919.995} C_VEL
LIN {X 0,Y 537.81,Z 720.175,A -85,B 0,C 180,E1 21918.51,E2 21918.51} C_VEL
LIN {X 0,Y 535.366,Z 748.209,A -85,B 0,C 180,E1 21917.936,E2 21917.936} C_VEL
LIN {X 0,Y 532.822,Z 769.704,A -85,B 0,C 180,E1 21917.345,E2 21917.345} C_VEL
LIN {X 0,Y 530.08,Z 789.185,A -85,B 0,C 180,E1 21916.689,E2 21916.689} C_VEL
LIN {X 0,Y 526.332,Z 812.485,A -85,B 0,C 180,E1 21915.741,E2 21915.741} C_VEL
LIN {X 0,Y 521.981,Z 835.6,A -85,B 0,C 180,E1 21914.592,E2 21914.592} C_VEL
LIN {X 0,Y 517.83,Z 855.588,A -85,B 0,C 180,E1 21913.425,E2 21913.425} C_VEL
LIN {X 0,Y 513.36,Z 875.704,A -85,B 0,C 180,E1 21912.068,E2 21912.068} C_VEL
LIN {X 0,Y 507.956,Z 898.254,A -85,B 0,C 180,E1 21910.288,E2 21910.288} C_VEL
LIN {X 0,Y 503.577,Z 915.603,A -85,B 0,C 180,E1 21908.709,E2 21908.709} C_VEL
LIN {X 0,Y 499.121,Z 932.841,A -85,B 0,C 180,E1 21906.935,E2 21906.935} C_VEL
LIN {X 0,Y 493.633,Z 953.596,A -85,B 0,C 180,E1 21904.471,E2 21904.471} C_VEL
LIN {X 0,Y 489.568,Z 969.064,A -85,B 0,C 180,E1 21902.351,E2 21902.351} C_VEL
LIN {X 0,Y 485.558,Z 984.925,A -85,B 0,C 180,E1 21899.89,E2 21899.89} C_VEL
LIN {X 0,Y 481.807,Z 1000.019,A -85,B 0,C 180,E1 21897.165,E2 21897.165} C_VEL
LIN {X 0,Y 479.196,Z 1011.52,A -85,B 0,C 180,E1 21894.797,E2 21894.797} C_VEL
LIN {X 0,Y 476.689,Z 1023.776,A -85,B 0,C 180,E1 21891.923,E2 21891.923} C_VEL
LIN {X 0,Y 474.755,Z 1034.459,A -85,B 0,C 180,E1 21888.926,E2 21888.926} C_VEL
LIN {X 0,Y 473.615,Z 1042.078,A -85,B 0,C 180,E1 21886.433,E2 21886.433} C_VEL
LIN {X 0,Y 472.759,Z 1049.463,A -85,B 0,C 180,E1 21883.578,E2 21883.578} C_VEL
LIN {X 0,Y 472.22,Z 1055.721,A -85,B 0,C 180,E1 21880.492,E2 21880.492} C_VEL
LIN {X 0,Y 472.024,Z 1059.711,A -85,B 0,C 180,E1 21877.914,E2 21877.914} C_VEL
LIN {X 0,Y 471.922,Z 1062.469,A -85,B 0,C 180,E1 21875.471,E2 21875.471} C_VEL
LIN {X 0,Y 471.914,Z 1064.36,A -85,B 0,C 180,E1 21872.793,E2 21872.793} C_VEL
LIN {X 0,Y 471.906,Z 1065.053,A -85,B 0,C 180,E1 21869.757,E2 21869.757} C_VEL
LIN {X 0,Y 471.914,Z 1064.225,A -85,B 0,C 180,E1 21866.964,E2 21866.964} C_VEL
LIN {X 0,Y 471.923,Z 1062.357,A -85,B 0,C 180,E1 21864.407,E2 21864.407} C_VEL
LIN {X 0,Y 472.029,Z 1059.555,A -85,B 0,C 180,E1 21861.963,E2 21861.963} C_VEL
LIN {X 0,Y 472.306,Z 1054.684,A -85,B 0,C 180,E1 21858.893,E2 21858.893} C_VEL
LIN {X 0,Y 472.921,Z 1047.939,A -85,B 0,C 180,E1 21855.803,E2 21855.803} C_VEL
LIN {X 0,Y 473.765,Z 1040.99,A -85,B 0,C 180,E1 21853.194,E2 21853.194} C_VEL
LIN {X 0,Y 475.253,Z 1031.525,A -85,B 0,C 180,E1 21850.201,E2 21850.201} C_VEL
LIN {X 0,Y 477.254,Z 1020.508,A -85,B 0,C 180,E1 21847.326,E2 21847.326} C_VEL
LIN {X 0,Y 479.402,Z 1010.082,A -85,B 0,C 180,E1 21844.951,E2 21844.951} C_VEL
LIN {X 0,Y 482.548,Z 996.371,A -85,B 0,C 180,E1 21842.211,E2 21842.211} C_VEL
LIN {X 0,Y 486.175,Z 981.088,A -85,B 0,C 180,E1 21839.607,E2 21839.607} C_VEL
LIN {X 0,Y 489.849,Z 966.352,A -85,B 0,C 180,E1 21837.393,E2 21837.393} C_VEL
LIN {X 0,Y 494.835,Z 946.777,A -85,B 0,C 180,E1 21834.839,E2 21834.839} C_VEL
LIN {X 0,Y 498.965,Z 930.322,A -85,B 0,C 180,E1 21832.974,E2 21832.974} C_VEL
LIN {X 0,Y 503.217,Z 913.169,A -85,B 0,C 180,E1 21831.252,E2 21831.252} C_VEL
LIN {X 0,Y 508.654,Z 890.266,A -85,B 0,C 180,E1 21829.26,E2 21829.26} C_VEL
LIN {X 0,Y 512.982,Z 870.943,A -85,B 0,C 180,E1 21827.818,E2 21827.818} C_VEL
LIN {X 0,Y 517.461,Z 849.674,A -85,B 0,C 180,E1 21826.437,E2 21826.437} C_VEL
LIN {X 0,Y 522.071,Z 825.296,A -85,B 0,C 180,E1 21825.109,E2 21825.109} C_VEL
LIN {X 0,Y 525.518,Z 804.785,A -85,B 0,C 180,E1 21824.168,E2 21824.168} C_VEL
LIN {X 0,Y 529.017,Z 781.349,A -85,B 0,C 180,E1 21823.268,E2 21823.268} C_VEL
LIN {X 0,Y 532.166,Z 755.219,A -85,B 0,C 180,E1 21822.484,E2 21822.484} C_VEL
LIN {X 0,Y 534.3,Z 733.126,A -85,B 0,C 180,E1 21821.977,E2 21821.977} C_VEL
LIN {X 0,Y 536.009,Z 706.509,A -85,B 0,C 180,E1 21821.514,E2 21821.514} C_VEL
LIN {X 0,Y 545.556,Z 472.585,A -85,B 0,C 180,E1 21818.04,E2 21818.04} C_VEL
LIN {X 0,Y 548.967,Z 389.725,A -85,B 0,C 180,E1 21816.783,E2 21816.783} C_VEL
LIN {X 0,Y 537.901,Z 371.788,A -85,B 0,C 180,E1 21814.862,E2 21814.862} C_VEL
LIN {X 0,Y 527.416,Z 355.69,A -85,B 0,C 180,E1 21812.899,E2 21812.899} C_VEL
LIN {X 0,Y 516.588,Z 340.105,A -85,B 0,C 180,E1 21810.698,E2 21810.698} C_VEL
LIN {X 0,Y 506.262,Z 326.087,A -85,B 0,C 180,E1 21808.392,E2 21808.392} C_VEL
LIN {X 0,Y 499.258,Z 317.11,A -85,B 0,C 180,E1 21806.687,E2 21806.687} C_VEL
LIN {X 0,Y 495.083,Z 311.958,A -85,B 0,C 180,E1 21805.608,E2 21805.608} C_VEL
LIN {X 0,Y 491.585,Z 308.169,A -85,B 0,C 180,E1 21804.676,E2 21804.676} C_VEL
LIN {X 0,Y 490.18,Z 306.07,A -85,B 0,C 180,E1 21804.27,E2 21804.27} C_VEL
LIN {X 0,Y 486.804,Z 302.881,A -85,B 0,C 180,E1 21803.323,E2 21803.323} C_VEL
LIN {X 0,Y 484.963,Z 299.913,A -85,B 0,C 180,E1 21802.742,E2 21802.742} C_VEL
LIN {X 0,Y 481.641,Z 297.282,A -85,B 0,C 180,E1 21801.751,E2 21801.751} C_VEL
LIN {X 0,Y 479.356,Z 293.502,A -85,B 0,C 180,E1 21800.961,E2 21800.961} C_VEL
LIN {X 0,Y 476.065,Z 291.292,A -85,B 0,C 180,E1 21799.892,E2 21799.892} C_VEL
LIN {X 0,Y 474.374,Z 288.338,A -85,B 0,C 180,E1 21799.226,E2 21799.226} C_VEL
LIN {X 0,Y 474.115,Z 287.022,A -85,B 0,C 180,E1 21798.752,E2 21798.752} C_VEL
LIN {X 0,Y 474.055,Z 286.913,A -85,B 0,C 180,E1 21795.287,E2 21795.287} C_VEL
LIN {X 0,Y 474.047,Z 286.907,A -85,B 0,C 180,E1 21791.683,E2 21791.683} C_VEL
LIN {X 0,Y 474.086,Z 286.895,A -85,B 0,C 180,E1 21788.246,E2 21788.246} C_VEL
LIN {X 0,Y 474.07,Z 286.9,A -85,B 0,C 180,E1 21784.84,E2 21784.84} C_VEL
LIN {X 0,Y 474.046,Z 286.918,A -85,B 0,C 180,E1 21781.329,E2 21781.329} C_VEL
LIN {X 0,Y 474.066,Z 286.931,A -85,B 0,C 180,E1 21777.824,E2 21777.824} C_VEL
LIN {X 0,Y 474.103,Z 286.908,A -85,B 0,C 180,E1 21774.19,E2 21774.19} C_VEL
LIN {X 0,Y 474.057,Z 286.899,A -85,B 0,C 180,E1 21770.776,E2 21770.776} C_VEL
LIN {X 0,Y 474.044,Z 286.9,A -85,B 0,C 180,E1 21767.204,E2 21767.204} C_VEL
LIN {X 0,Y 474.074,Z 286.902,A -85,B 0,C 180,E1 21763.709,E2 21763.709} C_VEL
LIN {X 0,Y 474.097,Z 286.905,A -85,B 0,C 180,E1 21760.15,E2 21760.15} C_VEL
LIN {X 0,Y 474.147,Z 287.147,A -85,B 0,C 180,E1 21757.953,E2 21757.953} C_VEL
LIN {X 0,Y 474.474,Z 288.618,A -85,B 0,C 180,E1 21757.545,E2 21757.545} C_VEL
LIN {X 0,Y 476.201,Z 291.455,A -85,B 0,C 180,E1 21756.88,E2 21756.88} C_VEL
LIN {X 0,Y 479.842,Z 294.061,A -85,B 0,C 180,E1 21755.698,E2 21755.698} C_VEL
LIN {X 0,Y 481.806,Z 297.406,A -85,B 0,C 180,E1 21755.019,E2 21755.019} C_VEL
LIN {X 0,Y 485.322,Z 300.275,A -85,B 0,C 180,E1 21753.97,E2 21753.97} C_VEL
LIN {X 0,Y 487.83,Z 304.069,A -85,B 0,C 180,E1 21753.197,E2 21753.197} C_VEL
LIN {X 0,Y 490.764,Z 306.767,A -85,B 0,C 180,E1 21752.386,E2 21752.386} C_VEL
LIN {X 0,Y 493.864,Z 310.913,A -85,B 0,C 180,E1 21751.523,E2 21751.523} C_VEL
LIN {X 0,Y 496.022,Z 313.04,A -85,B 0,C 180,E1 21750.967,E2 21750.967} C_VEL
LIN {X 0,Y 499.626,Z 317.481,A -85,B 0,C 180,E1 21750.045,E2 21750.045} C_VEL
LIN {X 0,Y 501.324,Z 319.428,A -85,B 0,C 180,E1 21749.628,E2 21749.628} C_VEL
LIN {X 0,Y 506.284,Z 325.601,A -85,B 0,C 180,E1 21748.442,E2 21748.442} C_VEL
LIN {X 0,Y 510.746,Z 331.203,A -85,B 0,C 180,E1 21747.427,E2 21747.427} C_VEL
LIN {X 0,Y 518.399,Z 340.946,A -85,B 0,C 180,E1 21745.788,E2 21745.788} C_VEL
LIN {X 0,Y 525.868,Z 351.057,A -85,B 0,C 180,E1 21744.286,E2 21744.286} C_VEL
LIN {X 0,Y 538.393,Z 369.83,A -85,B 0,C 180,E1 21741.933,E2 21741.933} C_VEL
LIN {X 0,Y 549.067,Z 387.103,A -85,B 0,C 180,E1 21740.076,E2 21740.076} C_VEL
LIN {X 0,Y 540.473,Z 592.031,A -85,B 0,C 180,E1 21737.015,E2 21737.015} C_VEL
LIN {X 0,Y 535.438,Z 712.775,A -85,B 0,C 180,E1 21735.207,E2 21735.207} C_VEL
LIN {X 0,Y 533.227,Z 740.165,A -85,B 0,C 180,E1 21734.65,E2 21734.65} C_VEL
LIN {X 0,Y 530.717,Z 762.819,A -85,B 0,C 180,E1 21734.023,E2 21734.023} C_VEL
LIN {X 0,Y 528.168,Z 782.115,A -85,B 0,C 180,E1 21733.367,E2 21733.367} C_VEL
LIN {X 0,Y 524.849,Z 803.911,A -85,B 0,C 180,E1 21732.482,E2 21732.482} C_VEL
LIN {X 0,Y 520.556,Z 828.16,A -85,B 0,C 180,E1 21731.284,E2 21731.284} C_VEL
LIN {X 0,Y 516.698,Z 847.678,A -85,B 0,C 180,E1 21730.147,E2 21730.147} C_VEL
LIN {X 0,Y 512.56,Z 867.157,A -85,B 0,C 180,E1 21728.842,E2 21728.842} C_VEL
LIN {X 0,Y 507.252,Z 890.334,A -85,B 0,C 180,E1 21727.028,E2 21727.028} C_VEL
LIN {X 0,Y 502.851,Z 908.419,A -85,B 0,C 180,E1 21725.386,E2 21725.386} C_VEL
LIN {X 0,Y 498.541,Z 925.68,A -85,B 0,C 180,E1 21723.611,E2 21723.611} C_VEL
LIN {X 0,Y 496.652,Z 932.999,A -85,B 0,C 180,E1 21722.785,E2 21722.785} C_VEL
LIN {X 0,Y 494.41,Z 938.512,A -85,B 0,C 180,E1 21722.2,E2 21722.2} C_VEL
LIN {X 0,Y 485.239,Z 953.101,A -85,B 0,C 180,E1 21720.752,E2 21720.752} C_VEL
LIN {X 0,Y 483.399,Z 957.394,A -85,B 0,C 180,E1 21720.194,E2 21720.194} C_VEL
LIN {X 0,Y 479.52,Z 971.952,A -85,B 0,C 180,E1 21717.98,E2 21717.98} C_VEL
LIN {X 0,Y 476.021,Z 985.565,A -85,B 0,C 180,E1 21715.639,E2 21715.639} C_VEL
LIN {X 0,Y 472.304,Z 1000.68,A -85,B 0,C 180,E1 21712.626,E2 21712.626} C_VEL
LIN {X 0,Y 469.918,Z 1011.316,A -85,B 0,C 180,E1 21710.163,E2 21710.163} C_VEL
LIN {X 0,Y 467.898,Z 1021.236,A -85,B 0,C 180,E1 21707.536,E2 21707.536} C_VEL
LIN {X 0,Y 466.109,Z 1031.553,A -85,B 0,C 180,E1 21704.282,E2 21704.282} C_VEL
LIN {X 0,Y 465.14,Z 1038.442,A -85,B 0,C 180,E1 21701.658,E2 21701.658} C_VEL
LIN {X 0,Y 464.522,Z 1044.151,A -85,B 0,C 180,E1 21699.04,E2 21699.04} C_VEL
LIN {X 0,Y 464.105,Z 1049.508,A -85,B 0,C 180,E1 21695.936,E2 21695.936} C_VEL
LIN {X 0,Y 463.948,Z 1053.002,A -85,B 0,C 180,E1 21692.965,E2 21692.965} C_VEL
LIN {X 0,Y 463.926,Z 1054.953,A -85,B 0,C 180,E1 21690.37,E2 21690.37} C_VEL
LIN {X 0,Y 463.906,Z 1055.821,A -85,B 0,C 180,E1 21687.9,E2 21687.9} C_VEL
LIN {X 0,Y 463.904,Z 1055.672,A -85,B 0,C 180,E1 21685.178,E2 21685.178} C_VEL
LIN {X 0,Y 463.923,Z 1054.032,A -85,B 0,C 180,E1 21682.071,E2 21682.071} C_VEL
LIN {X 0,Y 464.027,Z 1051.201,A -85,B 0,C 180,E1 21679.296,E2 21679.296} C_VEL
LIN {X 0,Y 464.231,Z 1047.427,A -85,B 0,C 180,E1 21676.676,E2 21676.676} C_VEL
LIN {X 0,Y 464.715,Z 1042.215,A -85,B 0,C 180,E1 21673.885,E2 21673.885} C_VEL
LIN {X 0,Y 465.716,Z 1034.258,A -85,B 0,C 180,E1 21670.562,E2 21670.562} C_VEL
LIN {X 0,Y 467.006,Z 1026.354,A -85,B 0,C 180,E1 21667.863,E2 21667.863} C_VEL
LIN {X 0,Y 468.808,Z 1017.103,A -85,B 0,C 180,E1 21665.155,E2 21665.155} C_VEL
LIN {X 0,Y 471.577,Z 1004.623,A -85,B 0,C 180,E1 21662.057,E2 21662.057} C_VEL
LIN {X 0,Y 474.513,Z 992.539,A -85,B 0,C 180,E1 21659.481,E2 21659.481} C_VEL
LIN {X 0,Y 478.361,Z 978.153,A -85,B 0,C 180,E1 21656.795,E2 21656.795} C_VEL
LIN {X 0,Y 482.644,Z 962.27,A -85,B 0,C 180,E1 21654.252,E2 21654.252} C_VEL
LIN {X 0,Y 486.705,Z 947.657,A -85,B 0,C 180,E1 21652.192,E2 21652.192} C_VEL
LIN {X 0,Y 491.81,Z 929.622,A -85,B 0,C 180,E1 21649.949,E2 21649.949} C_VEL
LIN {X 0,Y 497.109,Z 910.078,A -85,B 0,C 180,E1 21647.869,E2 21647.869} C_VEL
LIN {X 0,Y 501.475,Z 893.582,A -85,B 0,C 180,E1 21646.325,E2 21646.325} C_VEL
LIN {X 0,Y 506.282,Z 874.699,A -85,B 0,C 180,E1 21644.765,E2 21644.765} C_VEL
LIN {X 0,Y 511.73,Z 851.569,A -85,B 0,C 180,E1 21643.131,E2 21643.131} C_VEL
LIN {X 0,Y 515.924,Z 832.184,A -85,B 0,C 180,E1 21641.962,E2 21641.962} C_VEL
LIN {X 0,Y 519.704,Z 813.058,A -85,B 0,C 180,E1 21640.961,E2 21640.961} C_VEL
LIN {X 0,Y 524.074,Z 788.297,A -85,B 0,C 180,E1 21639.871,E2 21639.871} C_VEL
LIN {X 0,Y 527.416,Z 765.382,A -85,B 0,C 180,E1 21639.063,E2 21639.063} C_VEL
LIN {X 0,Y 530.014,Z 744.011,A -85,B 0,C 180,E1 21638.451,E2 21638.451} C_VEL
LIN {X 0,Y 532.538,Z 717.996,A -85,B 0,C 180,E1 21637.884,E2 21637.884} C_VEL
LIN {X 0,Y 534.952,Z 670.109,A -85,B 0,C 180,E1 21637.136,E2 21637.136} C_VEL
LIN {X 0,Y 545.263,Z 447.284,A -85,B 0,C 180,E1 21633.77,E2 21633.77} C_VEL
LIN {X 0,Y 547.823,Z 392.281,A -85,B 0,C 180,E1 21632.919,E2 21632.919} C_VEL
LIN {X 0,Y 537.373,Z 375.663,A -85,B 0,C 180,E1 21630.87,E2 21630.87} C_VEL
LIN {X 0,Y 526.118,Z 359.208,A -85,B 0,C 180,E1 21628.461,E2 21628.461} C_VEL
LIN {X 0,Y 518.029,Z 348.515,A -85,B 0,C 180,E1 21626.572,E2 21626.572} C_VEL
LIN {X 0,Y 512.341,Z 341.505,A -85,B 0,C 180,E1 21625.148,E2 21625.148} C_VEL
LIN {X 0,Y 508.849,Z 337.054,A -85,B 0,C 180,E1 21624.217,E2 21624.217} C_VEL
LIN {X 0,Y 504.632,Z 331.895,A -85,B 0,C 180,E1 21623.038,E2 21623.038} C_VEL
LIN {X 0,Y 500.795,Z 327.117,A -85,B 0,C 180,E1 21621.893,E2 21621.893} C_VEL
LIN {X 0,Y 496.653,Z 322.635,A -85,B 0,C 180,E1 21620.599,E2 21620.599} C_VEL
LIN {X 0,Y 495.128,Z 320.488,A -85,B 0,C 180,E1 21620.079,E2 21620.079} C_VEL
LIN {X 0,Y 491.667,Z 317.008,A -85,B 0,C 180,E1 21618.897,E2 21618.897} C_VEL
LIN {X 0,Y 489.829,Z 314.333,A -85,B 0,C 180,E1 21618.199,E2 21618.199} C_VEL
LIN {X 0,Y 486.413,Z 311.324,A -85,B 0,C 180,E1 21616.91,E2 21616.91} C_VEL
LIN {X 0,Y 484.472,Z 308.11,A -85,B 0,C 180,E1 21616.055,E2 21616.055} C_VEL
LIN {X 0,Y 480.883,Z 305.434,A -85,B 0,C 180,E1 21614.51,E2 21614.51} C_VEL
LIN {X 0,Y 478.891,Z 301.948,A -85,B 0,C 180,E1 21613.462,E2 21613.462} C_VEL
LIN {X 0,Y 474.309,Z 298.49,A -85,B 0,C 180,E1 21610.999,E2 21610.999} C_VEL
LIN {X 0,Y 472.372,Z 295.021,A -85,B 0,C 180,E1 21609.626,E2 21609.626} C_VEL
LIN {X 0,Y 467.782,Z 291.758,A -85,B 0,C 180,E1 21605.889,E2 21605.889} C_VEL
LIN {X 0,Y 466.275,Z 288.658,A -85,B 0,C 180,E1 21603.442,E2 21603.442} C_VEL
LIN {X 0,Y 466.109,Z 287.896,A -85,B 0,C 180,E1 21600.492,E2 21600.492} C_VEL
LIN {X 0,Y 466.116,Z 287.934,A -85,B 0,C 180,E1 21596.803,E2 21596.803} C_VEL
LIN {X 0,Y 466.306,Z 288.64,A -85,B 0,C 180,E1 21593.598,E2 21593.598} C_VEL
LIN {X 0,Y 468.935,Z 293.044,A -85,B 0,C 180,E1 21590.054,E2 21590.054} C_VEL
LIN {X 0,Y 472.632,Z 295.288,A -85,B 0,C 180,E1 21587.29,E2 21587.29} C_VEL
LIN {X 0,Y 474.607,Z 298.779,A -85,B 0,C 180,E1 21585.917,E2 21585.917} C_VEL
LIN {X 0,Y 477.959,Z 301.266,A -85,B 0,C 180,E1 21584.094,E2 21584.094} C_VEL
LIN {X 0,Y 478.937,Z 302.149,A -85,B 0,C 180,E1 21583.599,E2 21583.599} C_VEL
LIN {X 0,Y 480.89,Z 305.471,A -85,B 0,C 180,E1 21582.578,E2 21582.578} C_VEL
LIN {X 0,Y 484.75,Z 308.523,A -85,B 0,C 180,E1 21580.917,E2 21580.917} C_VEL
LIN {X 0,Y 487.436,Z 312.446,A -85,B 0,C 180,E1 21579.779,E2 21579.779} C_VEL
LIN {X 0,Y 490.389,Z 314.962,A -85,B 0,C 180,E1 21578.688,E2 21578.688} C_VEL
LIN {X 0,Y 493.335,Z 319.076,A -85,B 0,C 180,E1 21577.602,E2 21577.602} C_VEL
LIN {X 0,Y 495.819,Z 321.369,A -85,B 0,C 180,E1 21576.78,E2 21576.78} C_VEL
LIN {X 0,Y 499.158,Z 325.63,A -85,B 0,C 180,E1 21575.691,E2 21575.691} C_VEL
LIN {X 0,Y 501.274,Z 327.992,A -85,B 0,C 180,E1 21575.047,E2 21575.047} C_VEL
LIN {X 0,Y 508.418,Z 337.152,A -85,B 0,C 180,E1 21572.98,E2 21572.98} C_VEL
LIN {X 0,Y 516.605,Z 348.021,A -85,B 0,C 180,E1 21570.839,E2 21570.839} C_VEL
LIN {X 0,Y 525.775,Z 360.941,A -85,B 0,C 180,E1 21568.659,E2 21568.659} C_VEL
LIN {X 0,Y 535.87,Z 375.909,A -85,B 0,C 180,E1 21566.474,E2 21566.474} C_VEL
LIN {X 0,Y 546.572,Z 393.003,A -85,B 0,C 180,E1 21564.346,E2 21564.346} C_VEL
LIN {X 0,Y 547.903,Z 395.587,A -85,B 0,C 180,E1 21564.085,E2 21564.085} C_VEL
LIN {X 0,Y 537.069,Z 625.73,A -85,B 0,C 180,E1 21560.608,E2 21560.608} C_VEL
LIN {X 0,Y 532.647,Z 720.203,A -85,B 0,C 180,E1 21559.168,E2 21559.168} C_VEL
LIN {X 0,Y 530.118,Z 748.314,A -85,B 0,C 180,E1 21558.589,E2 21558.589} C_VEL
LIN {X 0,Y 527.535,Z 769.475,A -85,B 0,C 180,E1 21558.006,E2 21558.006} C_VEL
LIN {X 0,Y 524.609,Z 789.602,A -85,B 0,C 180,E1 21557.326,E2 21557.326} C_VEL
LIN {X 0,Y 520.533,Z 814.062,A -85,B 0,C 180,E1 21556.32,E2 21556.32} C_VEL
LIN {X 0,Y 516.04,Z 836.852,A -85,B 0,C 180,E1 21555.167,E2 21555.167} C_VEL
LIN {X 0,Y 511.953,Z 855.821,A -85,B 0,C 180,E1 21554.049,E2 21554.049} C_VEL
LIN {X 0,Y 506.966,Z 877.503,A -85,B 0,C 180,E1 21552.57,E2 21552.57} C_VEL
LIN {X 0,Y 501.549,Z 899.053,A -85,B 0,C 180,E1 21550.836,E2 21550.836} C_VEL
LIN {X 0,Y 496.985,Z 916.436,A -85,B 0,C 180,E1 21549.232,E2 21549.232} C_VEL
LIN {X 0,Y 491.975,Z 935.099,A -85,B 0,C 180,E1 21547.276,E2 21547.276} C_VEL
LIN {X 0,Y 486.62,Z 954.364,A -85,B 0,C 180,E1 21544.93,E2 21544.93} C_VEL
LIN {X 0,Y 482.565,Z 969.108,A -85,B 0,C 180,E1 21542.879,E2 21542.879} C_VEL
LIN {X 0,Y 478.167,Z 985.71,A -85,B 0,C 180,E1 21540.262,E2 21540.262} C_VEL
LIN {X 0,Y 474.419,Z 1000.023,A -85,B 0,C 180,E1 21537.624,E2 21537.624} C_VEL
LIN {X 0,Y 471.652,Z 1011.511,A -85,B 0,C 180,E1 21535.221,E2 21535.221} C_VEL
LIN {X 0,Y 468.997,Z 1023.799,A -85,B 0,C 180,E1 21532.289,E2 21532.289} C_VEL
LIN {X 0,Y 466.953,Z 1034.418,A -85,B 0,C 180,E1 21529.254,E2 21529.254} C_VEL
LIN {X 0,Y 465.741,Z 1042.027,A -85,B 0,C 180,E1 21526.719,E2 21526.719} C_VEL
LIN {X 0,Y 464.827,Z 1049.401,A -85,B 0,C 180,E1 21523.814,E2 21523.814} C_VEL
LIN {X 0,Y 464.249,Z 1055.648,A -85,B 0,C 180,E1 21520.674,E2 21520.674} C_VEL
LIN {X 0,Y 464.029,Z 1059.634,A -85,B 0,C 180,E1 21518.051,E2 21518.051} C_VEL
LIN {X 0,Y 463.922,Z 1062.391,A -85,B 0,C 180,E1 21515.566,E2 21515.566} C_VEL
LIN {X 0,Y 463.914,Z 1064.214,A -85,B 0,C 180,E1 21512.965,E2 21512.965} C_VEL
LIN {X 0,Y 463.908,Z 1064.998,A -85,B 0,C 180,E1 21509.877,E2 21509.877} C_VEL
LIN {X 0,Y 463.913,Z 1064.147,A -85,B 0,C 180,E1 21506.911,E2 21506.911} C_VEL
LIN {X 0,Y 463.925,Z 1062.279,A -85,B 0,C 180,E1 21504.31,E2 21504.31} C_VEL
LIN {X 0,Y 464.033,Z 1059.475,A -85,B 0,C 180,E1 21501.824,E2 21501.824} C_VEL
LIN {X 0,Y 464.333,Z 1054.598,A -85,B 0,C 180,E1 21498.699,E2 21498.699} C_VEL
LIN {X 0,Y 464.959,Z 1048.147,A -85,B 0,C 180,E1 21495.682,E2 21495.682} C_VEL
LIN {X 0,Y 465.789,Z 1041.595,A -85,B 0,C 180,E1 21493.154,E2 21493.154} C_VEL
LIN {X 0,Y 467.087,Z 1033.464,A -85,B 0,C 180,E1 21490.492,E2 21490.492} C_VEL
LIN {X 0,Y 469.385,Z 1021.409,A -85,B 0,C 180,E1 21487.189,E2 21487.189} C_VEL
LIN {X 0,Y 471.727,Z 1010.51,A -85,B 0,C 180,E1 21484.649,E2 21484.649} C_VEL
LIN {X 0,Y 474.839,Z 997.497,A -85,B 0,C 180,E1 21481.993,E2 21481.993} C_VEL
LIN {X 0,Y 478.783,Z 981.677,A -85,B 0,C 180,E1 21479.226,E2 21479.226} C_VEL
LIN {X 0,Y 482.418,Z 967.679,A -85,B 0,C 180,E1 21477.08,E2 21477.08} C_VEL
LIN {X 0,Y 487.259,Z 949.616,A -85,B 0,C 180,E1 21474.642,E2 21474.642} C_VEL
LIN {X 0,Y 492.048,Z 931.191,A -85,B 0,C 180,E1 21472.511,E2 21472.511} C_VEL
LIN {X 0,Y 496.441,Z 914.125,A -85,B 0,C 180,E1 21470.771,E2 21470.771} C_VEL
LIN {X 0,Y 501.733,Z 892.902,A -85,B 0,C 180,E1 21468.878,E2 21468.878} C_VEL
LIN {X 0,Y 506.528,Z 872.238,A -85,B 0,C 180,E1 21467.307,E2 21467.307} C_VEL
LIN {X 0,Y 510.651,Z 853.369,A -85,B 0,C 180,E1 21466.056,E2 21466.056} C_VEL
LIN {X 0,Y 515.293,Z 830.543,A -85,B 0,C 180,E1 21464.749,E2 21464.749} C_VEL
LIN {X 0,Y 519.436,Z 806.872,A -85,B 0,C 180,E1 21463.633,E2 21463.633} C_VEL
LIN {X 0,Y 522.697,Z 786.004,A -85,B 0,C 180,E1 21462.81,E2 21462.81} C_VEL
LIN {X 0,Y 526.055,Z 760.89,A -85,B 0,C 180,E1 21462.002,E2 21462.002} C_VEL
LIN {X 0,Y 528.607,Z 735.777,A -85,B 0,C 180,E1 21461.4,E2 21461.4} C_VEL
LIN {X 0,Y 530.217,Z 713.375,A -85,B 0,C 180,E1 21460.99,E2 21460.99} C_VEL
LIN {X 0,Y 540.238,Z 478.69,A -85,B 0,C 180,E1 21457.475,E2 21457.475} C_VEL
LIN {X 0,Y 543.933,Z 393.659,A -85,B 0,C 180,E1 21456.187,E2 21456.187} C_VEL
LIN {X 0,Y 533.827,Z 377.204,A -85,B 0,C 180,E1 21454.384,E2 21454.384} C_VEL
LIN {X 0,Y 524.105,Z 362.091,A -85,B 0,C 180,E1 21452.518,E2 21452.518} C_VEL
LIN {X 0,Y 513.176,Z 346.164,A -85,B 0,C 180,E1 21450.243,E2 21450.243} C_VEL
LIN {X 0,Y 503.325,Z 332.702,A -85,B 0,C 180,E1 21447.991,E2 21447.991} C_VEL
LIN {X 0,Y 496.835,Z 324.253,A -85,B 0,C 180,E1 21446.376,E2 21446.376} C_VEL
LIN {X 0,Y 492.699,Z 319.162,A -85,B 0,C 180,E1 21445.29,E2 21445.29} C_VEL
LIN {X 0,Y 489.068,Z 315.033,A -85,B 0,C 180,E1 21444.296,E2 21444.296} C_VEL
LIN {X 0,Y 487.655,Z 313.2,A -85,B 0,C 180,E1 21443.888,E2 21443.888} C_VEL
LIN {X 0,Y 484.274,Z 309.628,A -85,B 0,C 180,E1 21442.905,E2 21442.905} C_VEL
LIN {X 0,Y 482.702,Z 307.28,A -85,B 0,C 180,E1 21442.405,E2 21442.405} C_VEL
LIN {X 0,Y 479.37,Z 304.309,A -85,B 0,C 180,E1 21441.377,E2 21441.377} C_VEL
LIN {X 0,Y 477.531,Z 301.129,A -85,B 0,C 180,E1 21440.724,E2 21440.724} C_VEL
LIN {X 0,Y 474.128,Z 298.649,A -85,B 0,C 180,E1 21439.592,E2 21439.592} C_VEL
LIN {X 0,Y 472.137,Z 295.252,A -85,B 0,C 180,E1 21438.81,E2 21438.81} C_VEL
LIN {X 0,Y 471.123,Z 294.367,A -85,B 0,C 180,E1 21438.435,E2 21438.435} C_VEL
LIN {X 0,Y 468.06,Z 292.201,A -85,B 0,C 180,E1 21437.274,E2 21437.274} C_VEL
LIN {X 0,Y 466.268,Z 288.617,A -85,B 0,C 180,E1 21436.315,E2 21436.315} C_VEL
LIN {X 0,Y 466.113,Z 287.936,A -85,B 0,C 180,E1 21435.682,E2 21435.682} C_VEL
LIN {X 0,Y 466.142,Z 287.885,A -85,B 0,C 180,E1 21432.261,E2 21432.261} C_VEL
LIN {X 0,Y 466.156,Z 287.882,A -85,B 0,C 180,E1 21428.636,E2 21428.636} C_VEL
LIN {X 0,Y 466.112,Z 287.895,A -85,B 0,C 180,E1 21425.169,E2 21425.169} C_VEL
LIN {X 0,Y 466.109,Z 287.909,A -85,B 0,C 180,E1 21421.475,E2 21421.475} C_VEL
LIN {X 0,Y 466.144,Z 287.912,A -85,B 0,C 180,E1 21418.033,E2 21418.033} C_VEL
LIN {X 0,Y 466.161,Z 287.892,A -85,B 0,C 180,E1 21414.338,E2 21414.338} C_VEL
LIN {X 0,Y 466.113,Z 287.887,A -85,B 0,C 180,E1 21410.866,E2 21410.866} C_VEL
LIN {X 0,Y 466.105,Z 287.888,A -85,B 0,C 180,E1 21407.235,E2 21407.235} C_VEL
LIN {X 0,Y 466.145,Z 287.89,A -85,B 0,C 180,E1 21403.808,E2 21403.808} C_VEL
LIN {X 0,Y 466.13,Z 288.031,A -85,B 0,C 180,E1 21400.84,E2 21400.84} C_VEL
LIN {X 0,Y 466.493,Z 289.425,A -85,B 0,C 180,E1 21400.27,E2 21400.27} C_VEL
LIN {X 0,Y 468.326,Z 292.482,A -85,B 0,C 180,E1 21399.438,E2 21399.438} C_VEL
LIN {X 0,Y 471.597,Z 294.525,A -85,B 0,C 180,E1 21398.22,E2 21398.22} C_VEL
LIN {X 0,Y 472.398,Z 295.857,A -85,B 0,C 180,E1 21397.899,E2 21397.899} C_VEL
LIN {X 0,Y 474.439,Z 299.007,A -85,B 0,C 180,E1 21397.118,E2 21397.118} C_VEL
LIN {X 0,Y 477.767,Z 301.511,A -85,B 0,C 180,E1 21396.013,E2 21396.013} C_VEL
LIN {X 0,Y 480.154,Z 305.167,A -85,B 0,C 180,E1 21395.19,E2 21395.19} C_VEL
LIN {X 0,Y 483.254,Z 307.863,A -85,B 0,C 180,E1 21394.246,E2 21394.246} C_VEL
LIN {X 0,Y 486.133,Z 311.832,A -85,B 0,C 180,E1 21393.36,E2 21393.36} C_VEL
LIN {X 0,Y 488.547,Z 314.153,A -85,B 0,C 180,E1 21392.68,E2 21392.68} C_VEL
LIN {X 0,Y 491.924,Z 318.478,A -85,B 0,C 180,E1 21391.732,E2 21391.732} C_VEL
LIN {X 0,Y 493.745,Z 320.406,A -85,B 0,C 180,E1 21391.251,E2 21391.251} C_VEL
LIN {X 0,Y 497.641,Z 325.045,A -85,B 0,C 180,E1 21390.245,E2 21390.245} C_VEL
LIN {X 0,Y 503.799,Z 332.789,A -85,B 0,C 180,E1 21388.735,E2 21388.735} C_VEL
LIN {X 0,Y 508.55,Z 338.846,A -85,B 0,C 180,E1 21387.636,E2 21387.636} C_VEL
LIN {X 0,Y 515.658,Z 348.005,A -85,B 0,C 180,E1 21386.089,E2 21386.089} C_VEL
LIN {X 0,Y 523.44,Z 358.633,A -85,B 0,C 180,E1 21384.499,E2 21384.499} C_VEL
LIN {X 0,Y 536.894,Z 379.221,A -85,B 0,C 180,E1 21381.943,E2 21381.943} C_VEL
LIN {X 0,Y 543.97,Z 391.219,A -85,B 0,C 180,E1 21380.68,E2 21380.68} C_VEL
LIN {X 0,Y 535.092,Z 595.39,A -85,B 0,C 180,E1 21377.612,E2 21377.612} C_VEL
LIN {X 0,Y 530.01,Z 712.827,A -85,B 0,C 180,E1 21375.841,E2 21375.841} C_VEL
LIN {X 0,Y 527.747,Z 740.151,A -85,B 0,C 180,E1 21375.284,E2 21375.284} C_VEL
LIN {X 0,Y 525.165,Z 762.79,A -85,B 0,C 180,E1 21374.656,E2 21374.656} C_VEL
LIN {X 0,Y 522.456,Z 782.645,A -85,B 0,C 180,E1 21373.978,E2 21373.978} C_VEL
LIN {X 0,Y 518.798,Z 805.923,A -85,B 0,C 180,E1 21373.021,E2 21373.021} C_VEL
LIN {X 0,Y 514.561,Z 828.767,A -85,B 0,C 180,E1 21371.873,E2 21371.873} C_VEL
LIN {X 0,Y 510.696,Z 847.672,A -85,B 0,C 180,E1 21370.765,E2 21370.765} C_VEL
LIN {X 0,Y 506.303,Z 867.67,A -85,B 0,C 180,E1 21369.414,E2 21369.414} C_VEL
LIN {X 0,Y 500.975,Z 890.131,A -85,B 0,C 180,E1 21367.643,E2 21367.643} C_VEL
LIN {X 0,Y 496.491,Z 907.91,A -85,B 0,C 180,E1 21366.019,E2 21366.019} C_VEL
LIN {X 0,Y 492.195,Z 924.447,A -85,B 0,C 180,E1 21364.312,E2 21364.312} C_VEL
LIN {X 0,Y 487.02,Z 943.93,A -85,B 0,C 180,E1 21362.013,E2 21362.013} C_VEL
LIN {X 0,Y 483.399,Z 957.394,A -85,B 0,C 180,E1 21360.194,E2 21360.194} C_VEL
LIN {X 0,Y 481.173,Z 962.377,A -85,B 0,C 180,E1 21359.533,E2 21359.533} C_VEL
LIN {X 0,Y 472.13,Z 975.588,A -85,B 0,C 180,E1 21357.859,E2 21357.859} C_VEL
LIN {X 0,Y 470.388,Z 979.442,A -85,B 0,C 180,E1 21357.234,E2 21357.234} C_VEL
LIN {X 0,Y 466.77,Z 992.946,A -85,B 0,C 180,E1 21354.69,E2 21354.69} C_VEL
LIN {X 0,Y 463.857,Z 1004.724,A -85,B 0,C 180,E1 21352.162,E2 21352.162} C_VEL
LIN {X 0,Y 460.947,Z 1017.514,A -85,B 0,C 180,E1 21348.954,E2 21348.954} C_VEL
LIN {X 0,Y 459.158,Z 1026.432,A -85,B 0,C 180,E1 21346.315,E2 21346.315} C_VEL
LIN {X 0,Y 457.832,Z 1034.24,A -85,B 0,C 180,E1 21343.622,E2 21343.622} C_VEL
LIN {X 0,Y 456.771,Z 1042.311,A -85,B 0,C 180,E1 21340.213,E2 21340.213} C_VEL
LIN {X 0,Y 456.264,Z 1047.447,A -85,B 0,C 180,E1 21337.429,E2 21337.429} C_VEL
LIN {X 0,Y 456.044,Z 1051.062,A -85,B 0,C 180,E1 21334.905,E2 21334.905} C_VEL
LIN {X 0,Y 455.934,Z 1053.797,A -85,B 0,C 180,E1 21332.262,E2 21332.262} C_VEL
LIN {X 0,Y 455.911,Z 1055.683,A -85,B 0,C 180,E1 21329.12,E2 21329.12} C_VEL
LIN {X 0,Y 455.899,Z 1055.943,A -85,B 0,C 180,E1 21326.227,E2 21326.227} C_VEL
LIN {X 0,Y 455.918,Z 1055.159,A -85,B 0,C 180,E1 21323.704,E2 21323.704} C_VEL
LIN {X 0,Y 455.939,Z 1053.388,A -85,B 0,C 180,E1 21321.169,E2 21321.169} C_VEL
LIN {X 0,Y 456.066,Z 1050.614,A -85,B 0,C 180,E1 21318.62,E2 21318.62} C_VEL
LIN {X 0,Y 456.409,Z 1045.986,A -85,B 0,C 180,E1 21315.537,E2 21315.537} C_VEL
LIN {X 0,Y 457.156,Z 1039.341,A -85,B 0,C 180,E1 21312.301,E2 21312.301} C_VEL
LIN {X 0,Y 458.118,Z 1032.803,A -85,B 0,C 180,E1 21309.694,E2 21309.694} C_VEL
LIN {X 0,Y 459.675,Z 1024.268,A -85,B 0,C 180,E1 21306.814,E2 21306.814} C_VEL
LIN {X 0,Y 462.133,Z 1012.844,A -85,B 0,C 180,E1 21303.605,E2 21303.605} C_VEL
LIN {X 0,Y 464.687,Z 1002.217,A -85,B 0,C 180,E1 21301.044,E2 21301.044} C_VEL
LIN {X 0,Y 468.351,Z 988.589,A -85,B 0,C 180,E1 21298.175,E2 21298.175} C_VEL
LIN {X 0,Y 472.55,Z 973.389,A -85,B 0,C 180,E1 21295.454,E2 21295.454} C_VEL
LIN {X 0,Y 476.552,Z 959.542,A -85,B 0,C 180,E1 21293.274,E2 21293.274} C_VEL
LIN {X 0,Y 481.821,Z 941.71,A -85,B 0,C 180,E1 21290.809,E2 21290.809} C_VEL
LIN {X 0,Y 487.097,Z 923.255,A -85,B 0,C 180,E1 21288.625,E2 21288.625} C_VEL
LIN {X 0,Y 491.876,Z 906.361,A -85,B 0,C 180,E1 21286.868,E2 21286.868} C_VEL
LIN {X 0,Y 497.744,Z 884.789,A -85,B 0,C 180,E1 21284.918,E2 21284.918} C_VEL
LIN {X 0,Y 502.799,Z 864.798,A -85,B 0,C 180,E1 21283.377,E2 21283.377} C_VEL
LIN {X 0,Y 507.434,Z 845.224,A -85,B 0,C 180,E1 21282.065,E2 21282.065} C_VEL
LIN {X 0,Y 512.765,Z 820.554,A -85,B 0,C 180,E1 21280.664,E2 21280.664} C_VEL
LIN {X 0,Y 516.823,Z 798.993,A -85,B 0,C 180,E1 21279.646,E2 21279.646} C_VEL
LIN {X 0,Y 520.349,Z 777.898,A -85,B 0,C 180,E1 21278.813,E2 21278.813} C_VEL
LIN {X 0,Y 524.012,Z 751.468,A -85,B 0,C 180,E1 21277.973,E2 21277.973} C_VEL
LIN {X 0,Y 526.519,Z 728.18,A -85,B 0,C 180,E1 21277.418,E2 21277.418} C_VEL
LIN {X 0,Y 528.258,Z 705.289,A -85,B 0,C 180,E1 21276.999,E2 21276.999} C_VEL
LIN {X 0,Y 539.52,Z 470.322,A -85,B 0,C 180,E1 21273.431,E2 21273.431} C_VEL
LIN {X 0,Y 543.109,Z 396.345,A -85,B 0,C 180,E1 21272.287,E2 21272.287} C_VEL
LIN {X 0,Y 533.573,Z 381.238,A -85,B 0,C 180,E1 21270.365,E2 21270.365} C_VEL
LIN {X 0,Y 523.165,Z 365.766,A -85,B 0,C 180,E1 21268.076,E2 21268.076} C_VEL
LIN {X 0,Y 515.286,Z 355.294,A -85,B 0,C 180,E1 21266.197,E2 21266.197} C_VEL
LIN {X 0,Y 506.723,Z 344.404,A -85,B 0,C 180,E1 21263.954,E2 21263.954} C_VEL
LIN {X 0,Y 502.186,Z 338.89,A -85,B 0,C 180,E1 21262.661,E2 21262.661} C_VEL
LIN {X 0,Y 497.97,Z 333.736,A -85,B 0,C 180,E1 21261.373,E2 21261.373} C_VEL
LIN {X 0,Y 494.241,Z 329.333,A -85,B 0,C 180,E1 21260.161,E2 21260.161} C_VEL
LIN {X 0,Y 493.001,Z 327.802,A -85,B 0,C 180,E1 21259.736,E2 21259.736} C_VEL
LIN {X 0,Y 489.476,Z 323.93,A -85,B 0,C 180,E1 21258.49,E2 21258.49} C_VEL
LIN {X 0,Y 488.256,Z 322.034,A -85,B 0,C 180,E1 21258.013,E2 21258.013} C_VEL
LIN {X 0,Y 484.741,Z 318.859,A -85,B 0,C 180,E1 21256.662,E2 21256.662} C_VEL
LIN {X 0,Y 482.678,Z 315.687,A -85,B 0,C 180,E1 21255.746,E2 21255.746} C_VEL
LIN {X 0,Y 479.182,Z 312.827,A -85,B 0,C 180,E1 21254.193,E2 21254.193} C_VEL
LIN {X 0,Y 477.116,Z 309.31,A -85,B 0,C 180,E1 21253.081,E2 21253.081} C_VEL
LIN {X 0,Y 473.328,Z 306.626,A -85,B 0,C 180,E1 21251.022,E2 21251.022} C_VEL
LIN {X 0,Y 471.536,Z 303.526,A -85,B 0,C 180,E1 21249.767,E2 21249.767} C_VEL
LIN {X 0,Y 470.701,Z 302.574,A -85,B 0,C 180,E1 21249.167,E2 21249.167} C_VEL
LIN {X 0,Y 466.692,Z 299.635,A -85,B 0,C 180,E1 21245.779,E2 21245.779} C_VEL
LIN {X 0,Y 464.968,Z 296.508,A -85,B 0,C 180,E1 21243.329,E2 21243.329} C_VEL
LIN {X 0,Y 463.6,Z 295.459,A -85,B 0,C 180,E1 21239.876,E2 21239.876} C_VEL
LIN {X 0,Y 464.464,Z 296.008,A -85,B 0,C 180,E1 21234.689,E2 21234.689} C_VEL
LIN {X 0,Y 465.302,Z 297.071,A -85,B 0,C 180,E1 21233.212,E2 21233.212} C_VEL
LIN {X 0,Y 467.968,Z 301.034,A -85,B 0,C 180,E1 21230.034,E2 21230.034} C_VEL
LIN {X 0,Y 471.401,Z 303.113,A -85,B 0,C 180,E1 21227.443,E2 21227.443} C_VEL
LIN {X 0,Y 473.159,Z 306.366,A -85,B 0,C 180,E1 21226.185,E2 21226.185} C_VEL
LIN {X 0,Y 476.542,Z 309.036,A -85,B 0,C 180,E1 21224.296,E2 21224.296} C_VEL
LIN {X 0,Y 477.395,Z 309.786,A -85,B 0,C 180,E1 21223.857,E2 21223.857} C_VEL
LIN {X 0,Y 479.558,Z 313.304,A -85,B 0,C 180,E1 21222.715,E2 21222.715} C_VEL
LIN {X 0,Y 483.104,Z 316.174,A -85,B 0,C 180,E1 21221.163,E2 21221.163} C_VEL
LIN {X 0,Y 486.048,Z 320.293,A -85,B 0,C 180,E1 21219.907,E2 21219.907} C_VEL
LIN {X 0,Y 488.661,Z 322.638,A -85,B 0,C 180,E1 21218.923,E2 21218.923} C_VEL
LIN {X 0,Y 491.744,Z 326.783,A -85,B 0,C 180,E1 21217.777,E2 21217.777} C_VEL
LIN {X 0,Y 493.948,Z 328.915,A -85,B 0,C 180,E1 21217.034,E2 21217.034} C_VEL
LIN {X 0,Y 497.514,Z 333.345,A -85,B 0,C 180,E1 21215.859,E2 21215.859} C_VEL
LIN {X 0,Y 499.853,Z 336.237,A -85,B 0,C 180,E1 21215.129,E2 21215.129} C_VEL
LIN {X 0,Y 506.12,Z 344.319,A -85,B 0,C 180,E1 21213.292,E2 21213.292} C_VEL
